LIN {X 0,Y 152.112,Z 664.807,A -85,B 0,C 180,E1 -25600.837,E2 -25600.837} C_VEL
LIN {X 0,Y 146.265,Z 675.889,A -85,B 0,C 180,E1 -25603.884,E2 -25603.884} C_VEL
LIN {X 0,Y 140.329,Z 686.128,A -85,B 0,C 180,E1 -25607.459,E2 -25607.459} C_VEL
LIN {X 0,Y 134.268,Z 696.183,A -85,B 0,C 180,E1 -25612.046,E2 -25612.046} C_VEL
LIN {X 0,Y 129.23,Z 704.605,A -85,B 0,C 180,E1 -25617.054,E2 -25617.054} C_VEL
LIN {X 0,Y 124.936,Z 712.522,A -85,B 0,C 180,E1 -25623.254,E2 -25623.254} C_VEL
LIN {X 0,Y 122.172,Z 718.854,A -85,B 0,C 180,E1 -25629.808,E2 -25629.808} C_VEL
LIN {X 0,Y 121.041,Z 723.776,A -85,B 0,C 180,E1 -25636.569,E2 -25636.569} C_VEL
LIN {X 0,Y 121.369,Z 727.342,A -85,B 0,C 180,E1 -25643.348,E2 -25643.348} C_VEL
LIN {X 0,Y 121.7,Z 728.339,A -85,B 0,C 180,E1 -25646.011,E2 -25646.011} C_VEL
LIN {X 0,Y 121.232,Z 728.844,A -85,B 0,C 180,E1 -25647.815,E2 -25647.815} C_VEL
LIN {X 0,Y 119.721,Z 729.035,A -85,B 0,C 180,E1 -25649.561,E2 -25649.561} C_VEL
LIN {X 0,Y 114.837,Z 728.936,A -85,B 0,C 180,E1 -25654.372,E2 -25654.372} C_VEL
LIN {X 0,Y 114.337,Z 728.882,A -85,B 0,C 180,E1 -25655.721,E2 -25655.721} C_VEL
LIN {X 0,Y 113.821,Z 728.676,A -85,B 0,C 180,E1 -25660.673,E2 -25660.673} C_VEL
LIN {X 0,Y 114.375,Z 727.382,A -85,B 0,C 180,E1 -25667.891,E2 -25667.891} C_VEL
LIN {X 0,Y 117.287,Z 724.46,A -85,B 0,C 180,E1 -25675.999,E2 -25675.999} C_VEL
LIN {X 0,Y 122.084,Z 720.301,A -85,B 0,C 180,E1 -25683.151,E2 -25683.151} C_VEL
LIN {X 0,Y 128.148,Z 715.223,A -85,B 0,C 180,E1 -25689.099,E2 -25689.099} C_VEL
LIN {X 0,Y 135.57,Z 708.791,A -85,B 0,C 180,E1 -25694.412,E2 -25694.412} C_VEL
LIN {X 0,Y 144.175,Z 700.89,A -85,B 0,C 180,E1 -25699.071,E2 -25699.071} C_VEL
LIN {X 0,Y 153.874,Z 691.31,A -85,B 0,C 180,E1 -25703.059,E2 -25703.059} C_VEL
LIN {X 0,Y 161.553,Z 682.701,A -85,B 0,C 180,E1 -25705.742,E2 -25705.742} C_VEL
LIN {X 0,Y 169.66,Z 672.712,A -85,B 0,C 180,E1 -25708.12,E2 -25708.12} C_VEL
LIN {X 0,Y 178.185,Z 660.946,A -85,B 0,C 180,E1 -25710.191,E2 -25710.191} C_VEL
LIN {X 0,Y 186.287,Z 648.041,A -85,B 0,C 180,E1 -25711.863,E2 -25711.863} C_VEL
LIN {X 0,Y 193.002,Z 635.336,A -85,B 0,C 180,E1 -25713.14,E2 -25713.14} C_VEL
LIN {X 0,Y 198.339,Z 623.513,A -85,B 0,C 180,E1 -25714.041,E2 -25714.041} C_VEL
LIN {X 0,Y 203.672,Z 608.798,A -85,B 0,C 180,E1 -25714.925,E2 -25714.925} C_VEL
LIN {X 0,Y 207.856,Z 593.51,A -85,B 0,C 180,E1 -25715.612,E2 -25715.612} C_VEL
LIN {X 0,Y 210.78,Z 577.845,A -85,B 0,C 180,E1 -25716.128,E2 -25716.128} C_VEL
LIN {X 0,Y 214.688,Z 540.152,A -85,B 0,C 180,E1 -25717.041,E2 -25717.041} C_VEL
LIN {X 0,Y 212.531,Z 531.894,A -85,B 0,C 180,E1 -25719.647,E2 -25719.647} C_VEL
LIN {X 0,Y 210.604,Z 524.936,A -85,B 0,C 180,E1 -25722.358,E2 -25722.358} C_VEL
LIN {X 0,Y 208.889,Z 519.075,A -85,B 0,C 180,E1 -25725.299,E2 -25725.299} C_VEL
LIN {X 0,Y 207.864,Z 515.191,A -85,B 0,C 180,E1 -25727.626,E2 -25727.626} C_VEL
LIN {X 0,Y 206.577,Z 509.756,A -85,B 0,C 180,E1 -25732.318,E2 -25732.318} C_VEL
LIN {X 0,Y 206.426,Z 508.775,A -85,B 0,C 180,E1 -25733.504,E2 -25733.504} C_VEL
LIN {X 0,Y 206.448,Z 508.658,A -85,B 0,C 180,E1 -25739.513,E2 -25739.513} C_VEL
LIN {X 0,Y 208.229,Z 512.983,A -85,B 0,C 180,E1 -25745.508,E2 -25745.508} C_VEL
LIN {X 0,Y 210.191,Z 517.111,A -85,B 0,C 180,E1 -25749.042,E2 -25749.042} C_VEL
LIN {X 0,Y 212.228,Z 521.339,A -85,B 0,C 180,E1 -25751.824,E2 -25751.824} C_VEL
LIN {X 0,Y 215.125,Z 527.412,A -85,B 0,C 180,E1 -25755.015,E2 -25755.015} C_VEL
LIN {X 0,Y 215.758,Z 528.889,A -85,B 0,C 180,E1 -25755.648,E2 -25755.648} C_VEL
LIN {X 0,Y 213.115,Z 556.855,A -85,B 0,C 180,E1 -25756.59,E2 -25756.59} C_VEL
LIN {X 0,Y 210.858,Z 570.576,A -85,B 0,C 180,E1 -25757.266,E2 -25757.266} C_VEL
LIN {X 0,Y 207.171,Z 585.652,A -85,B 0,C 180,E1 -25758.227,E2 -25758.227} C_VEL
LIN {X 0,Y 202.935,Z 598.669,A -85,B 0,C 180,E1 -25759.322,E2 -25759.322} C_VEL
LIN {X 0,Y 197.926,Z 611.211,A -85,B 0,C 180,E1 -25760.677,E2 -25760.677} C_VEL
LIN {X 0,Y 191.785,Z 623.736,A -85,B 0,C 180,E1 -25762.293,E2 -25762.293} C_VEL
LIN {X 0,Y 184.944,Z 635.502,A -85,B 0,C 180,E1 -25764.22,E2 -25764.22} C_VEL
LIN {X 0,Y 176.984,Z 647.191,A -85,B 0,C 180,E1 -25766.693,E2 -25766.693} C_VEL
LIN {X 0,Y 169.299,Z 656.934,A -85,B 0,C 180,E1 -25769.341,E2 -25769.341} C_VEL
LIN {X 0,Y 160.734,Z 666.373,A -85,B 0,C 180,E1 -25772.685,E2 -25772.685} C_VEL
LIN {X 0,Y 152.46,Z 674.345,A -85,B 0,C 180,E1 -25776.451,E2 -25776.451} C_VEL
LIN {X 0,Y 144.183,Z 681.32,A -85,B 0,C 180,E1 -25780.932,E2 -25780.932} C_VEL
LIN {X 0,Y 136.527,Z 686.987,A -85,B 0,C 180,E1 -25786.112,E2 -25786.112} C_VEL
LIN {X 0,Y 131.621,Z 690.179,A -85,B 0,C 180,E1 -25790.155,E2 -25790.155} C_VEL
LIN {X 0,Y 125.932,Z 693.387,A -85,B 0,C 180,E1 -25796.079,E2 -25796.079} C_VEL
LIN {X 0,Y 121.441,Z 695.394,A -85,B 0,C 180,E1 -25802.423,E2 -25802.423} C_VEL
LIN {X 0,Y 118.353,Z 696.242,A -85,B 0,C 180,E1 -25809.129,E2 -25809.129} C_VEL
LIN {X 0,Y 116.654,Z 695.972,A -85,B 0,C 180,E1 -25816.057,E2 -25816.057} C_VEL
LIN {X 0,Y 116.026,Z 694.601,A -85,B 0,C 180,E1 -25823.043,E2 -25823.043} C_VEL
LIN {X 0,Y 116.863,Z 692.077,A -85,B 0,C 180,E1 -25830.001,E2 -25830.001} C_VEL
LIN {X 0,Y 118.905,Z 688.408,A -85,B 0,C 180,E1 -25836.79,E2 -25836.79} C_VEL
LIN {X 0,Y 122.063,Z 683.523,A -85,B 0,C 180,E1 -25843.316,E2 -25843.316} C_VEL
LIN {X 0,Y 126.468,Z 677.262,A -85,B 0,C 180,E1 -25849.478,E2 -25849.478} C_VEL
LIN {X 0,Y 131.942,Z 669.449,A -85,B 0,C 180,E1 -25855.223,E2 -25855.223} C_VEL
LIN {X 0,Y 137.496,Z 661.145,A -85,B 0,C 180,E1 -25859.892,E2 -25859.892} C_VEL
LIN {X 0,Y 143.772,Z 651.153,A -85,B 0,C 180,E1 -25864.205,E2 -25864.205} C_VEL
LIN {X 0,Y 149.59,Z 640.955,A -85,B 0,C 180,E1 -25867.645,E2 -25867.645} C_VEL
LIN {X 0,Y 155.595,Z 628.801,A -85,B 0,C 180,E1 -25870.915,E2 -25870.915} C_VEL
LIN {X 0,Y 161.011,Z 616.564,A -85,B 0,C 180,E1 -25873.43,E2 -25873.43} C_VEL
LIN {X 0,Y 166.031,Z 603.169,A -85,B 0,C 180,E1 -25875.586,E2 -25875.586} C_VEL
LIN {X 0,Y 170.263,Z 589.275,A -85,B 0,C 180,E1 -25877.328,E2 -25877.328} C_VEL
LIN {X 0,Y 173.623,Z 575.007,A -85,B 0,C 180,E1 -25878.71,E2 -25878.71} C_VEL
LIN {X 0,Y 176.335,Z 559.317,A -85,B 0,C 180,E1 -25879.769,E2 -25879.769} C_VEL
LIN {X 0,Y 177.885,Z 543.275,A -85,B 0,C 180,E1 -25880.541,E2 -25880.541} C_VEL
LIN {X 0,Y 181.077,Z 501.444,A -85,B 0,C 180,E1 -25882,E2 -25882} C_VEL
LIN {X 0,Y 176.773,Z 492.406,A -85,B 0,C 180,E1 -25885.022,E2 -25885.022} C_VEL
LIN {X 0,Y 172.294,Z 483.86,A -85,B 0,C 180,E1 -25888.613,E2 -25888.613} C_VEL
LIN {X 0,Y 168.158,Z 476.667,A -85,B 0,C 180,E1 -25892.541,E2 -25892.541} C_VEL
LIN {X 0,Y 165.346,Z 472.291,A -85,B 0,C 180,E1 -25895.716,E2 -25895.716} C_VEL
LIN {X 0,Y 163.231,Z 468.887,A -85,B 0,C 180,E1 -25898.6,E2 -25898.6} C_VEL
LIN {X 0,Y 160.878,Z 465.055,A -85,B 0,C 180,E1 -25902.718,E2 -25902.718} C_VEL
LIN {X 0,Y 158.454,Z 461.541,A -85,B 0,C 180,E1 -25910.004,E2 -25910.004} C_VEL
LIN {X 0,Y 158.278,Z 459.994,A -85,B 0,C 180,E1 -25912.344,E2 -25912.344} C_VEL
LIN {X 0,Y 158.418,Z 459.872,A -85,B 0,C 180,E1 -25917.616,E2 -25917.616} C_VEL
LIN {X 0,Y 159.139,Z 462.833,A -85,B 0,C 180,E1 -25921.897,E2 -25921.897} C_VEL
LIN {X 0,Y 160.93,Z 464.889,A -85,B 0,C 180,E1 -25926.25,E2 -25926.25} C_VEL
LIN {X 0,Y 163.185,Z 468.728,A -85,B 0,C 180,E1 -25930.233,E2 -25930.233} C_VEL
LIN {X 0,Y 164.069,Z 470.08,A -85,B 0,C 180,E1 -25931.504,E2 -25931.504} C_VEL
LIN {X 0,Y 165.979,Z 474.343,A -85,B 0,C 180,E1 -25934.11,E2 -25934.11} C_VEL
LIN {X 0,Y 168.676,Z 480.782,A -85,B 0,C 180,E1 -25937.269,E2 -25937.269} C_VEL
LIN {X 0,Y 171.447,Z 487.752,A -85,B 0,C 180,E1 -25940.078,E2 -25940.078} C_VEL
LIN {X 0,Y 174.742,Z 497.166,A -85,B 0,C 180,E1 -25943.077,E2 -25943.077} C_VEL
LIN {X 0,Y 178.052,Z 507.617,A -85,B 0,C 180,E1 -25945.807,E2 -25945.807} C_VEL
LIN {X 0,Y 178.78,Z 510.414,A -85,B 0,C 180,E1 -25946.404,E2 -25946.404} C_VEL
LIN {X 0,Y 178.869,Z 533.313,A -85,B 0,C 180,E1 -25948.131,E2 -25948.131} C_VEL
LIN {X 0,Y 174.573,Z 581.759,A -85,B 0,C 180,E1 -25949.655,E2 -25949.655} C_VEL
LIN {X 0,Y 171.96,Z 597.666,A -85,B 0,C 180,E1 -25950.453,E2 -25950.453} C_VEL
LIN {X 0,Y 168.411,Z 612.372,A -85,B 0,C 180,E1 -25951.474,E2 -25951.474} C_VEL
LIN {X 0,Y 164.078,Z 626.316,A -85,B 0,C 180,E1 -25952.797,E2 -25952.797} C_VEL
LIN {X 0,Y 158.843,Z 639.968,A -85,B 0,C 180,E1 -25954.507,E2 -25954.507} C_VEL
LIN {X 0,Y 152.428,Z 653.818,A -85,B 0,C 180,E1 -25956.759,E2 -25956.759} C_VEL
LIN {X 0,Y 146.345,Z 665.337,A -85,B 0,C 180,E1 -25959.251,E2 -25959.251} C_VEL
LIN {X 0,Y 140.291,Z 676.167,A -85,B 0,C 180,E1 -25962.361,E2 -25962.361} C_VEL
LIN {X 0,Y 134.108,Z 686.187,A -85,B 0,C 180,E1 -25966.023,E2 -25966.023} C_VEL
LIN {X 0,Y 127.627,Z 696.341,A -85,B 0,C 180,E1 -25970.926,E2 -25970.926} C_VEL
LIN {X 0,Y 121.908,Z 705.397,A -85,B 0,C 180,E1 -25976.792,E2 -25976.792} C_VEL
LIN {X 0,Y 117.648,Z 712.863,A -85,B 0,C 180,E1 -25983.269,E2 -25983.269} C_VEL
LIN {X 0,Y 114.906,Z 718.974,A -85,B 0,C 180,E1 -25990.342,E2 -25990.342} C_VEL
LIN {X 0,Y 114.027,Z 722.601,A -85,B 0,C 180,E1 -25995.726,E2 -25995.726} C_VEL
LIN {X 0,Y 114.263,Z 726.206,A -85,B 0,C 180,E1 -26002.933,E2 -26002.933} C_VEL
LIN {X 0,Y 115.499,Z 728.454,A -85,B 0,C 180,E1 -26009.999,E2 -26009.999} C_VEL
LIN {X 0,Y 114.337,Z 728.882,A -85,B 0,C 180,E1 -26015.721,E2 -26015.721} C_VEL
LIN {X 0,Y 113.784,Z 728.846,A -85,B 0,C 180,E1 -26017.676,E2 -26017.676} C_VEL
LIN {X 0,Y 111.621,Z 728.326,A -85,B 0,C 180,E1 -26021.535,E2 -26021.535} C_VEL
LIN {X 0,Y 108.362,Z 726.846,A -85,B 0,C 180,E1 -26027.486,E2 -26027.486} C_VEL
LIN {X 0,Y 108.015,Z 725.981,A -85,B 0,C 180,E1 -26030.593,E2 -26030.593} C_VEL
LIN {X 0,Y 108.244,Z 725.674,A -85,B 0,C 180,E1 -26031.623,E2 -26031.623} C_VEL
LIN {X 0,Y 110.575,Z 723.732,A -85,B 0,C 180,E1 -26037.151,E2 -26037.151} C_VEL
LIN {X 0,Y 116.1,Z 719.409,A -85,B 0,C 180,E1 -26045.102,E2 -26045.102} C_VEL
LIN {X 0,Y 122.646,Z 714.362,A -85,B 0,C 180,E1 -26051.22,E2 -26051.22} C_VEL
LIN {X 0,Y 130.523,Z 707.987,A -85,B 0,C 180,E1 -26056.624,E2 -26056.624} C_VEL
LIN {X 0,Y 138.396,Z 701.205,A -85,B 0,C 180,E1 -26060.749,E2 -26060.749} C_VEL
LIN {X 0,Y 148.374,Z 691.91,A -85,B 0,C 180,E1 -26064.789,E2 -26064.789} C_VEL
LIN {X 0,Y 156.505,Z 683.356,A -85,B 0,C 180,E1 -26067.559,E2 -26067.559} C_VEL
LIN {X 0,Y 166.001,Z 672.212,A -85,B 0,C 180,E1 -26070.212,E2 -26070.212} C_VEL
LIN {X 0,Y 174.758,Z 660.554,A -85,B 0,C 180,E1 -26072.215,E2 -26072.215} C_VEL
LIN {X 0,Y 183.045,Z 647.785,A -85,B 0,C 180,E1 -26073.824,E2 -26073.824} C_VEL
LIN {X 0,Y 189.897,Z 635.255,A -85,B 0,C 180,E1 -26075.053,E2 -26075.053} C_VEL
LIN {X 0,Y 195.343,Z 623.545,A -85,B 0,C 180,E1 -26075.909,E2 -26075.909} C_VEL
LIN {X 0,Y 200.78,Z 609.126,A -85,B 0,C 180,E1 -26076.752,E2 -26076.752} C_VEL
LIN {X 0,Y 205.041,Z 594.319,A -85,B 0,C 180,E1 -26077.409,E2 -26077.409} C_VEL
LIN {X 0,Y 208.127,Z 579.032,A -85,B 0,C 180,E1 -26077.911,E2 -26077.911} C_VEL
LIN {X 0,Y 210.906,Z 554.927,A -85,B 0,C 180,E1 -26078.497,E2 -26078.497} C_VEL
LIN {X 0,Y 212.063,Z 543.415,A -85,B 0,C 180,E1 -26078.775,E2 -26078.775} C_VEL
LIN {X 0,Y 210.048,Z 535.02,A -85,B 0,C 180,E1 -26081.604,E2 -26081.604} C_VEL
LIN {X 0,Y 208.705,Z 529.937,A -85,B 0,C 180,E1 -26083.782,E2 -26083.782} C_VEL
LIN {X 0,Y 207.452,Z 525.087,A -85,B 0,C 180,E1 -26086.282,E2 -26086.282} C_VEL
LIN {X 0,Y 206.613,Z 521.553,A -85,B 0,C 180,E1 -26088.473,E2 -26088.473} C_VEL
LIN {X 0,Y 205.649,Z 516.707,A -85,B 0,C 180,E1 -26092.588,E2 -26092.588} C_VEL
LIN {X 0,Y 205.456,Z 515.784,A -85,B 0,C 180,E1 -26094.11,E2 -26094.11} C_VEL
LIN {X 0,Y 205.5,Z 515.62,A -85,B 0,C 180,E1 -26099.021,E2 -26099.021} C_VEL
LIN {X 0,Y 205.929,Z 517.273,A -85,B 0,C 180,E1 -26101.62,E2 -26101.62} C_VEL
LIN {X 0,Y 207.132,Z 519.832,A -85,B 0,C 180,E1 -26105.08,E2 -26105.08} C_VEL
LIN {X 0,Y 208.816,Z 523.632,A -85,B 0,C 180,E1 -26108.349,E2 -26108.349} C_VEL
LIN {X 0,Y 210.833,Z 528.018,A -85,B 0,C 180,E1 -26111.287,E2 -26111.287} C_VEL
LIN {X 0,Y 213.11,Z 533.062,A -85,B 0,C 180,E1 -26113.975,E2 -26113.975} C_VEL
LIN {X 0,Y 210.566,Z 558.418,A -85,B 0,C 180,E1 -26114.827,E2 -26114.827} C_VEL
LIN {X 0,Y 208.164,Z 572.425,A -85,B 0,C 180,E1 -26115.528,E2 -26115.528} C_VEL
LIN {X 0,Y 204.652,Z 586.243,A -85,B 0,C 180,E1 -26116.389,E2 -26116.389} C_VEL
LIN {X 0,Y 200.295,Z 599.365,A -85,B 0,C 180,E1 -26117.461,E2 -26117.461} C_VEL
LIN {X 0,Y 194.771,Z 612.768,A -85,B 0,C 180,E1 -26118.872,E2 -26118.872} C_VEL
LIN {X 0,Y 189.111,Z 623.995,A -85,B 0,C 180,E1 -26120.28,E2 -26120.28} C_VEL
LIN {X 0,Y 182.104,Z 635.823,A -85,B 0,C 180,E1 -26122.15,E2 -26122.15} C_VEL
LIN {X 0,Y 173.868,Z 647.633,A -85,B 0,C 180,E1 -26124.571,E2 -26124.571} C_VEL
LIN {X 0,Y 165.884,Z 657.476,A -85,B 0,C 180,E1 -26127.169,E2 -26127.169} C_VEL
LIN {X 0,Y 158.226,Z 665.783,A -85,B 0,C 180,E1 -26129.992,E2 -26129.992} C_VEL
LIN {X 0,Y 149.708,Z 673.835,A -85,B 0,C 180,E1 -26133.568,E2 -26133.568} C_VEL
LIN {X 0,Y 141.732,Z 680.433,A -85,B 0,C 180,E1 -26137.501,E2 -26137.501} C_VEL
LIN {X 0,Y 133.469,Z 686.463,A -85,B 0,C 180,E1 -26142.511,E2 -26142.511} C_VEL
LIN {X 0,Y 126.179,Z 691.039,A -85,B 0,C 180,E1 -26148.061,E2 -26148.061} C_VEL
LIN {X 0,Y 120.042,Z 694.301,A -85,B 0,C 180,E1 -26154.167,E2 -26154.167} C_VEL
LIN {X 0,Y 115.137,Z 696.359,A -85,B 0,C 180,E1 -26160.772,E2 -26160.772} C_VEL
LIN {X 0,Y 111.693,Z 697.26,A -85,B 0,C 180,E1 -26167.821,E2 -26167.821} C_VEL
LIN {X 0,Y 109.743,Z 697.031,A -85,B 0,C 180,E1 -26175.159,E2 -26175.159} C_VEL
LIN {X 0,Y 108.988,Z 695.69,A -85,B 0,C 180,E1 -26182.592,E2 -26182.592} C_VEL
LIN {X 0,Y 109.794,Z 693.218,A -85,B 0,C 180,E1 -26190.001,E2 -26190.001} C_VEL
LIN {X 0,Y 111.922,Z 689.6,A -85,B 0,C 180,E1 -26197.216,E2 -26197.216} C_VEL
LIN {X 0,Y 115.242,Z 684.772,A -85,B 0,C 180,E1 -26204.12,E2 -26204.12} C_VEL
LIN {X 0,Y 119.905,Z 678.569,A -85,B 0,C 180,E1 -26210.591,E2 -26210.591} C_VEL
LIN {X 0,Y 125.651,Z 670.828,A -85,B 0,C 180,E1 -26216.581,E2 -26216.581} C_VEL
LIN {X 0,Y 131.5,Z 662.597,A -85,B 0,C 180,E1 -26221.406,E2 -26221.406} C_VEL
LIN {X 0,Y 138.059,Z 652.696,A -85,B 0,C 180,E1 -26225.833,E2 -26225.833} C_VEL
LIN {X 0,Y 144.136,Z 642.602,A -85,B 0,C 180,E1 -26229.337,E2 -26229.337} C_VEL
LIN {X 0,Y 150.417,Z 630.569,A -85,B 0,C 180,E1 -26232.648,E2 -26232.648} C_VEL
LIN {X 0,Y 156.035,Z 618.496,A -85,B 0,C 180,E1 -26235.186,E2 -26235.186} C_VEL
LIN {X 0,Y 161.262,Z 605.302,A -85,B 0,C 180,E1 -26237.343,E2 -26237.343} C_VEL
LIN {X 0,Y 165.643,Z 591.684,A -85,B 0,C 180,E1 -26239.091,E2 -26239.091} C_VEL
LIN {X 0,Y 169.131,Z 577.782,A -85,B 0,C 180,E1 -26240.474,E2 -26240.474} C_VEL
LIN {X 0,Y 171.984,Z 562.633,A -85,B 0,C 180,E1 -26241.553,E2 -26241.553} C_VEL
LIN {X 0,Y 173.766,Z 547.313,A -85,B 0,C 180,E1 -26242.31,E2 -26242.31} C_VEL
LIN {X 0,Y 176.966,Z 507.169,A -85,B 0,C 180,E1 -26243.726,E2 -26243.726} C_VEL
LIN {X 0,Y 177.068,Z 504.448,A -85,B 0,C 180,E1 -26243.885,E2 -26243.885} C_VEL
LIN {X 0,Y 173.15,Z 496.062,A -85,B 0,C 180,E1 -26246.92,E2 -26246.92} C_VEL
LIN {X 0,Y 169.353,Z 488.56,A -85,B 0,C 180,E1 -26250.289,E2 -26250.289} C_VEL
LIN {X 0,Y 165.766,Z 482.228,A -85,B 0,C 180,E1 -26254.026,E2 -26254.026} C_VEL
LIN {X 0,Y 163.781,Z 478.872,A -85,B 0,C 180,E1 -26256.467,E2 -26256.467} C_VEL
LIN {X 0,Y 161.727,Z 475.429,A -85,B 0,C 180,E1 -26259.457,E2 -26259.457} C_VEL
LIN {X 0,Y 159.517,Z 471.62,A -85,B 0,C 180,E1 -26263.687,E2 -26263.687} C_VEL
LIN {X 0,Y 157.609,Z 468.874,A -85,B 0,C 180,E1 -26269.725,E2 -26269.725} C_VEL
LIN {X 0,Y 157.362,Z 467.006,A -85,B 0,C 180,E1 -26272.945,E2 -26272.945} C_VEL
LIN {X 0,Y 157.502,Z 467.081,A -85,B 0,C 180,E1 -26277.442,E2 -26277.442} C_VEL
LIN {X 0,Y 158.254,Z 469.982,A -85,B 0,C 180,E1 -26281.908,E2 -26281.908} C_VEL
LIN {X 0,Y 159.761,Z 471.82,A -85,B 0,C 180,E1 -26285.728,E2 -26285.728} C_VEL
LIN {X 0,Y 161.89,Z 475.532,A -85,B 0,C 180,E1 -26289.684,E2 -26289.684} C_VEL
LIN {X 0,Y 163.035,Z 477.817,A -85,B 0,C 180,E1 -26291.46,E2 -26291.46} C_VEL
LIN {X 0,Y 164.162,Z 480.658,A -85,B 0,C 180,E1 -26293.106,E2 -26293.106} C_VEL
LIN {X 0,Y 166.379,Z 486.256,A -85,B 0,C 180,E1 -26295.936,E2 -26295.936} C_VEL
LIN {X 0,Y 169.023,Z 493.456,A -85,B 0,C 180,E1 -26298.877,E2 -26298.877} C_VEL
LIN {X 0,Y 171.838,Z 502.041,A -85,B 0,C 180,E1 -26301.676,E2 -26301.676} C_VEL
LIN {X 0,Y 175.081,Z 513.049,A -85,B 0,C 180,E1 -26304.595,E2 -26304.595} C_VEL
LIN {X 0,Y 174.908,Z 535.394,A -85,B 0,C 180,E1 -26306.266,E2 -26306.266} C_VEL
LIN {X 0,Y 170.777,Z 580.315,A -85,B 0,C 180,E1 -26307.655,E2 -26307.655} C_VEL
LIN {X 0,Y 168.047,Z 596.417,A -85,B 0,C 180,E1 -26308.43,E2 -26308.43} C_VEL
LIN {X 0,Y 164.413,Z 611.138,A -85,B 0,C 180,E1 -26309.431,E2 -26309.431} C_VEL
LIN {X 0,Y 160.298,Z 624.113,A -85,B 0,C 180,E1 -26310.636,E2 -26310.636} C_VEL
LIN {X 0,Y 154.899,Z 638.009,A -85,B 0,C 180,E1 -26312.324,E2 -26312.324} C_VEL
LIN {X 0,Y 148.631,Z 651.257,A -85,B 0,C 180,E1 -26314.4,E2 -26314.4} C_VEL
LIN {X 0,Y 141.884,Z 663.665,A -85,B 0,C 180,E1 -26316.992,E2 -26316.992} C_VEL
LIN {X 0,Y 135.513,Z 674.596,A -85,B 0,C 180,E1 -26320.096,E2 -26320.096} C_VEL
LIN {X 0,Y 129.022,Z 684.714,A -85,B 0,C 180,E1 -26323.801,E2 -26323.801} C_VEL
LIN {X 0,Y 123.209,Z 693.309,A -85,B 0,C 180,E1 -26327.862,E2 -26327.862} C_VEL
LIN {X 0,Y 117.382,Z 701.932,A -85,B 0,C 180,E1 -26333.22,E2 -26333.22} C_VEL
LIN {X 0,Y 112.19,Z 709.964,A -85,B 0,C 180,E1 -26339.923,E2 -26339.923} C_VEL
LIN {X 0,Y 108.725,Z 716.409,A -85,B 0,C 180,E1 -26347.179,E2 -26347.179} C_VEL
LIN {X 0,Y 107.026,Z 721.409,A -85,B 0,C 180,E1 -26354.771,E2 -26354.771} C_VEL
LIN {X 0,Y 107.142,Z 725.065,A -85,B 0,C 180,E1 -26362.46,E2 -26362.46} C_VEL
LIN {X 0,Y 108.393,Z 727.372,A -85,B 0,C 180,E1 -26369.999,E2 -26369.999} C_VEL
LIN {X 0,Y 107.083,Z 727.865,A -85,B 0,C 180,E1 -26377.541,E2 -26377.541} C_VEL
LIN {X 0,Y 106.902,Z 727.158,A -85,B 0,C 180,E1 -26385.244,E2 -26385.244} C_VEL
LIN {X 0,Y 108.244,Z 725.674,A -85,B 0,C 180,E1 -26391.623,E2 -26391.623} C_VEL
LIN {X 0,Y 108.72,Z 724.686,A -85,B 0,C 180,E1 -26394.691,E2 -26394.691} C_VEL
LIN {X 0,Y 108.395,Z 722.594,A -85,B 0,C 180,E1 -26399.809,E2 -26399.809} C_VEL
LIN {X 0,Y 108.624,Z 720.558,A -85,B 0,C 180,E1 -26403.868,E2 -26403.868} C_VEL
LIN {X 0,Y 109.916,Z 718.836,A -85,B 0,C 180,E1 -26406.758,E2 -26406.758} C_VEL
LIN {X 0,Y 110.658,Z 718.231,A -85,B 0,C 180,E1 -26407.654,E2 -26407.654} C_VEL
LIN {X 0,Y 117.317,Z 713.505,A -85,B 0,C 180,E1 -26413.542,E2 -26413.542} C_VEL
LIN {X 0,Y 125.684,Z 707.187,A -85,B 0,C 180,E1 -26419.012,E2 -26419.012} C_VEL
LIN {X 0,Y 135.238,Z 699.421,A -85,B 0,C 180,E1 -26423.654,E2 -26423.654} C_VEL
LIN {X 0,Y 144.38,Z 691.245,A -85,B 0,C 180,E1 -26427.102,E2 -26427.102} C_VEL
LIN {X 0,Y 152.598,Z 682.98,A -85,B 0,C 180,E1 -26429.762,E2 -26429.762} C_VEL
LIN {X 0,Y 161.119,Z 673.488,A -85,B 0,C 180,E1 -26432.038,E2 -26432.038} C_VEL
LIN {X 0,Y 170.797,Z 661.236,A -85,B 0,C 180,E1 -26434.168,E2 -26434.168} C_VEL
LIN {X 0,Y 179.248,Z 648.81,A -85,B 0,C 180,E1 -26435.721,E2 -26435.721} C_VEL
LIN {X 0,Y 187.016,Z 635.164,A -85,B 0,C 180,E1 -26437.023,E2 -26437.023} C_VEL
LIN {X 0,Y 192.564,Z 623.575,A -85,B 0,C 180,E1 -26437.831,E2 -26437.831} C_VEL
LIN {X 0,Y 198.093,Z 609.452,A -85,B 0,C 180,E1 -26438.633,E2 -26438.633} C_VEL
LIN {X 0,Y 202.628,Z 594.364,A -85,B 0,C 180,E1 -26439.285,E2 -26439.285} C_VEL
LIN {X 0,Y 205.909,Z 578.826,A -85,B 0,C 180,E1 -26439.784,E2 -26439.784} C_VEL
LIN {X 0,Y 208.479,Z 557.906,A -85,B 0,C 180,E1 -26440.285,E2 -26440.285} C_VEL
LIN {X 0,Y 209.647,Z 546.785,A -85,B 0,C 180,E1 -26440.528,E2 -26440.528} C_VEL
LIN {X 0,Y 207.883,Z 538.858,A -85,B 0,C 180,E1 -26443.419,E2 -26443.419} C_VEL
LIN {X 0,Y 206.241,Z 531.798,A -85,B 0,C 180,E1 -26446.866,E2 -26446.866} C_VEL
LIN {X 0,Y 205.418,Z 527.904,A -85,B 0,C 180,E1 -26449.31,E2 -26449.31} C_VEL
LIN {X 0,Y 204.675,Z 523.442,A -85,B 0,C 180,E1 -26453.208,E2 -26453.208} C_VEL
LIN {X 0,Y 204.589,Z 522.852,A -85,B 0,C 180,E1 -26454.085,E2 -26454.085} C_VEL
LIN {X 0,Y 204.66,Z 522.742,A -85,B 0,C 180,E1 -26459.263,E2 -26459.263} C_VEL
LIN {X 0,Y 206.043,Z 526.707,A -85,B 0,C 180,E1 -26464.647,E2 -26464.647} C_VEL
LIN {X 0,Y 207.551,Z 530.322,A -85,B 0,C 180,E1 -26467.785,E2 -26467.785} C_VEL
LIN {X 0,Y 209.656,Z 535.161,A -85,B 0,C 180,E1 -26471.014,E2 -26471.014} C_VEL
LIN {X 0,Y 210.607,Z 537.691,A -85,B 0,C 180,E1 -26472.276,E2 -26472.276} C_VEL
LIN {X 0,Y 208.197,Z 560.164,A -85,B 0,C 180,E1 -26473.034,E2 -26473.034} C_VEL
LIN {X 0,Y 205.63,Z 574.297,A -85,B 0,C 180,E1 -26473.741,E2 -26473.741} C_VEL
LIN {X 0,Y 201.971,Z 588.128,A -85,B 0,C 180,E1 -26474.59,E2 -26474.59} C_VEL
LIN {X 0,Y 197.133,Z 602.066,A -85,B 0,C 180,E1 -26475.732,E2 -26475.732} C_VEL
LIN {X 0,Y 191.228,Z 615.598,A -85,B 0,C 180,E1 -26477.155,E2 -26477.155} C_VEL
LIN {X 0,Y 184.595,Z 627.95,A -85,B 0,C 180,E1 -26478.735,E2 -26478.735} C_VEL
LIN {X 0,Y 177.471,Z 639.17,A -85,B 0,C 180,E1 -26480.561,E2 -26480.561} C_VEL
LIN {X 0,Y 169.605,Z 649.838,A -85,B 0,C 180,E1 -26482.788,E2 -26482.788} C_VEL
LIN {X 0,Y 161.414,Z 659.44,A -85,B 0,C 180,E1 -26485.349,E2 -26485.349} C_VEL
LIN {X 0,Y 152.15,Z 668.832,A -85,B 0,C 180,E1 -26488.646,E2 -26488.646} C_VEL
LIN {X 0,Y 144.623,Z 675.552,A -85,B 0,C 180,E1 -26491.747,E2 -26491.747} C_VEL
LIN {X 0,Y 135.2,Z 682.857,A -85,B 0,C 180,E1 -26496.324,E2 -26496.324} C_VEL
LIN {X 0,Y 128.708,Z 687.265,A -85,B 0,C 180,E1 -26500.145,E2 -26500.145} C_VEL
LIN {X 0,Y 120.932,Z 691.899,A -85,B 0,C 180,E1 -26505.786,E2 -26505.786} C_VEL
LIN {X 0,Y 114.292,Z 695.217,A -85,B 0,C 180,E1 -26512.057,E2 -26512.057} C_VEL
LIN {X 0,Y 108.939,Z 697.326,A -85,B 0,C 180,E1 -26518.931,E2 -26518.931} C_VEL
LIN {X 0,Y 105.117,Z 698.277,A -85,B 0,C 180,E1 -26526.352,E2 -26526.352} C_VEL
LIN {X 0,Y 102.864,Z 698.076,A -85,B 0,C 180,E1 -26534.142,E2 -26534.142} C_VEL
LIN {X 0,Y 101.96,Z 696.779,A -85,B 0,C 180,E1 -26542.078,E2 -26542.078} C_VEL
LIN {X 0,Y 102.729,Z 694.356,A -85,B 0,C 180,E1 -26550.002,E2 -26550.002} C_VEL
LIN {X 0,Y 104.947,Z 690.789,A -85,B 0,C 180,E1 -26557.698,E2 -26557.698} C_VEL
LIN {X 0,Y 108.446,Z 686.017,A -85,B 0,C 180,E1 -26565.025,E2 -26565.025} C_VEL
LIN {X 0,Y 113.367,Z 679.875,A -85,B 0,C 180,E1 -26571.837,E2 -26571.837} C_VEL
LIN {X 0,Y 119.437,Z 672.199,A -85,B 0,C 180,E1 -26578.083,E2 -26578.083} C_VEL
LIN {X 0,Y 125.6,Z 664.041,A -85,B 0,C 180,E1 -26583.064,E2 -26583.064} C_VEL
LIN {X 0,Y 132.472,Z 654.228,A -85,B 0,C 180,E1 -26587.598,E2 -26587.598} C_VEL
LIN {X 0,Y 138.834,Z 644.223,A -85,B 0,C 180,E1 -26591.154,E2 -26591.154} C_VEL
LIN {X 0,Y 145.4,Z 632.32,A -85,B 0,C 180,E1 -26594.497,E2 -26594.497} C_VEL
LIN {X 0,Y 151.212,Z 620.368,A -85,B 0,C 180,E1 -26597.056,E2 -26597.056} C_VEL
LIN {X 0,Y 156.626,Z 607.354,A -85,B 0,C 180,E1 -26599.218,E2 -26599.218} C_VEL
LIN {X 0,Y 161.484,Z 593.017,A -85,B 0,C 180,E1 -26601.073,E2 -26601.073} C_VEL
LIN {X 0,Y 165.426,Z 577.946,A -85,B 0,C 180,E1 -26602.553,E2 -26602.553} C_VEL
LIN {X 0,Y 168.409,Z 562.39,A -85,B 0,C 180,E1 -26603.617,E2 -26603.617} C_VEL
LIN {X 0,Y 170.178,Z 546.885,A -85,B 0,C 180,E1 -26604.362,E2 -26604.362} C_VEL
LIN {X 0,Y 173.343,Z 507.8,A -85,B 0,C 180,E1 -26605.774,E2 -26605.774} C_VEL
LIN {X 0,Y 169.281,Z 498.823,A -85,B 0,C 180,E1 -26609.305,E2 -26609.305} C_VEL
LIN {X 0,Y 166.035,Z 492.321,A -85,B 0,C 180,E1 -26612.58,E2 -26612.58} C_VEL
LIN {X 0,Y 162.659,Z 486.034,A -85,B 0,C 180,E1 -26616.682,E2 -26616.682} C_VEL
LIN {X 0,Y 160.349,Z 482.108,A -85,B 0,C 180,E1 -26620.181,E2 -26620.181} C_VEL
LIN {X 0,Y 158.377,Z 478.512,A -85,B 0,C 180,E1 -26624.228,E2 -26624.228} C_VEL
LIN {X 0,Y 156.635,Z 475.708,A -85,B 0,C 180,E1 -26630.34,E2 -26630.34} C_VEL
LIN {X 0,Y 156.466,Z 474.001,A -85,B 0,C 180,E1 -26633.552,E2 -26633.552} C_VEL
LIN {X 0,Y 156.593,Z 474.269,A -85,B 0,C 180,E1 -26637.276,E2 -26637.276} C_VEL
LIN {X 0,Y 157.37,Z 477.122,A -85,B 0,C 180,E1 -26641.919,E2 -26641.919} C_VEL
LIN {X 0,Y 158.563,Z 478.622,A -85,B 0,C 180,E1 -26645.085,E2 -26645.085} C_VEL
LIN {X 0,Y 160.972,Z 483.055,A -85,B 0,C 180,E1 -26649.74,E2 -26649.74} C_VEL
LIN {X 0,Y 162.272,Z 486.508,A -85,B 0,C 180,E1 -26651.871,E2 -26651.871} C_VEL
LIN {X 0,Y 164.307,Z 492.109,A -85,B 0,C 180,E1 -26654.741,E2 -26654.741} C_VEL
LIN {X 0,Y 166.726,Z 499.277,A -85,B 0,C 180,E1 -26657.695,E2 -26657.695} C_VEL
LIN {X 0,Y 169.426,Z 508.237,A -85,B 0,C 180,E1 -26660.625,E2 -26660.625} C_VEL
LIN {X 0,Y 171.556,Z 516.284,A -85,B 0,C 180,E1 -26662.764,E2 -26662.764} C_VEL
LIN {X 0,Y 171.229,Z 536.211,A -85,B 0,C 180,E1 -26664.268,E2 -26664.268} C_VEL
LIN {X 0,Y 167.019,Z 579.936,A -85,B 0,C 180,E1 -26665.607,E2 -26665.607} C_VEL
LIN {X 0,Y 164.23,Z 595.762,A -85,B 0,C 180,E1 -26666.365,E2 -26666.365} C_VEL
LIN {X 0,Y 160.294,Z 611.04,A -85,B 0,C 180,E1 -26667.397,E2 -26667.397} C_VEL
LIN {X 0,Y 156.059,Z 623.907,A -85,B 0,C 180,E1 -26668.578,E2 -26668.578} C_VEL
LIN {X 0,Y 150.498,Z 637.643,A -85,B 0,C 180,E1 -26670.241,E2 -26670.241} C_VEL
LIN {X 0,Y 143.622,Z 651.56,A -85,B 0,C 180,E1 -26672.424,E2 -26672.424} C_VEL
LIN {X 0,Y 136.417,Z 664.191,A -85,B 0,C 180,E1 -26675.13,E2 -26675.13} C_VEL
LIN {X 0,Y 128.658,Z 676.669,A -85,B 0,C 180,E1 -26678.884,E2 -26678.884} C_VEL
LIN {X 0,Y 121.983,Z 686.312,A -85,B 0,C 180,E1 -26682.728,E2 -26682.728} C_VEL
LIN {X 0,Y 115.108,Z 695.83,A -85,B 0,C 180,E1 -26687.808,E2 -26687.808} C_VEL
LIN {X 0,Y 109.303,Z 703.772,A -85,B 0,C 180,E1 -26693.504,E2 -26693.504} C_VEL
LIN {X 0,Y 104.729,Z 710.571,A -85,B 0,C 180,E1 -26700.003,E2 -26700.003} C_VEL
LIN {X 0,Y 101.401,Z 716.524,A -85,B 0,C 180,E1 -26707.591,E2 -26707.591} C_VEL
LIN {X 0,Y 99.893,Z 721.246,A -85,B 0,C 180,E1 -26715.743,E2 -26715.743} C_VEL
LIN {X 0,Y 100.025,Z 723.922,A -85,B 0,C 180,E1 -26721.92,E2 -26721.92} C_VEL
LIN {X 0,Y 101.285,Z 726.288,A -85,B 0,C 180,E1 -26729.998,E2 -26729.998} C_VEL
LIN {X 0,Y 100.521,Z 726.711,A -85,B 0,C 180,E1 -26734.008,E2 -26734.008} C_VEL
LIN {X 0,Y 99.722,Z 726.622,A -85,B 0,C 180,E1 -26742.204,E2 -26742.204} C_VEL
LIN {X 0,Y 100.742,Z 725.394,A -85,B 0,C 180,E1 -26750.412,E2 -26750.412} C_VEL
LIN {X 0,Y 103.933,Z 722.95,A -85,B 0,C 180,E1 -26758.472,E2 -26758.472} C_VEL
LIN {X 0,Y 110.282,Z 718.509,A -85,B 0,C 180,E1 -26767.255,E2 -26767.255} C_VEL
LIN {X 0,Y 110.658,Z 718.231,A -85,B 0,C 180,E1 -26767.654,E2 -26767.654} C_VEL
LIN {X 0,Y 112.664,Z 716.386,A -85,B 0,C 180,E1 -26770.338,E2 -26770.338} C_VEL
LIN {X 0,Y 114.893,Z 712.97,A -85,B 0,C 180,E1 -26774.898,E2 -26774.898} C_VEL
LIN {X 0,Y 117.767,Z 709.211,A -85,B 0,C 180,E1 -26779.185,E2 -26779.185} C_VEL
LIN {X 0,Y 120.666,Z 706.701,A -85,B 0,C 180,E1 -26781.348,E2 -26781.348} C_VEL
LIN {X 0,Y 129.801,Z 699.734,A -85,B 0,C 180,E1 -26785.655,E2 -26785.655} C_VEL
LIN {X 0,Y 139.227,Z 691.844,A -85,B 0,C 180,E1 -26789.103,E2 -26789.103} C_VEL
LIN {X 0,Y 148.934,Z 682.6,A -85,B 0,C 180,E1 -26792.076,E2 -26792.076} C_VEL
LIN {X 0,Y 157.899,Z 672.941,A -85,B 0,C 180,E1 -26794.326,E2 -26794.326} C_VEL
LIN {X 0,Y 167.827,Z 660.803,A -85,B 0,C 180,E1 -26796.349,E2 -26796.349} C_VEL
LIN {X 0,Y 176.444,Z 648.487,A -85,B 0,C 180,E1 -26797.826,E2 -26797.826} C_VEL
LIN {X 0,Y 184.361,Z 635.004,A -85,B 0,C 180,E1 -26799.055,E2 -26799.055} C_VEL
LIN {X 0,Y 190.811,Z 621.834,A -85,B 0,C 180,E1 -26799.915,E2 -26799.915} C_VEL
LIN {X 0,Y 196.426,Z 607.523,A -85,B 0,C 180,E1 -26800.673,E2 -26800.673} C_VEL
LIN {X 0,Y 200.966,Z 592.392,A -85,B 0,C 180,E1 -26801.278,E2 -26801.278} C_VEL
LIN {X 0,Y 204.17,Z 577.144,A -85,B 0,C 180,E1 -26801.738,E2 -26801.738} C_VEL
LIN {X 0,Y 206.928,Z 554.742,A -85,B 0,C 180,E1 -26802.234,E2 -26802.234} C_VEL
LIN {X 0,Y 207.384,Z 550.17,A -85,B 0,C 180,E1 -26802.37,E2 -26802.37} C_VEL
LIN {X 0,Y 206.007,Z 543.205,A -85,B 0,C 180,E1 -26805.089,E2 -26805.089} C_VEL
LIN {X 0,Y 204.853,Z 537.548,A -85,B 0,C 180,E1 -26808.032,E2 -26808.032} C_VEL
LIN {X 0,Y 204.325,Z 534.604,A -85,B 0,C 180,E1 -26809.91,E2 -26809.91} C_VEL
LIN {X 0,Y 203.728,Z 530.188,A -85,B 0,C 180,E1 -26813.812,E2 -26813.812} C_VEL
LIN {X 0,Y 203.697,Z 529.672,A -85,B 0,C 180,E1 -26818.567,E2 -26818.567} C_VEL
LIN {X 0,Y 204.877,Z 533.236,A -85,B 0,C 180,E1 -26823.935,E2 -26823.935} C_VEL
LIN {X 0,Y 206.328,Z 537.069,A -85,B 0,C 180,E1 -26827.255,E2 -26827.255} C_VEL
LIN {X 0,Y 208.176,Z 541.617,A -85,B 0,C 180,E1 -26830.306,E2 -26830.306} C_VEL
LIN {X 0,Y 208.329,Z 542.017,A -85,B 0,C 180,E1 -26830.531,E2 -26830.531} C_VEL
LIN {X 0,Y 206.012,Z 562.102,A -85,B 0,C 180,E1 -26831.215,E2 -26831.215} C_VEL
LIN {X 0,Y 203.287,Z 576.239,A -85,B 0,C 180,E1 -26831.924,E2 -26831.924} C_VEL
LIN {X 0,Y 199.883,Z 588.74,A -85,B 0,C 180,E1 -26832.666,E2 -26832.666} C_VEL
LIN {X 0,Y 195.29,Z 601.76,A -85,B 0,C 180,E1 -26833.682,E2 -26833.682} C_VEL
LIN {X 0,Y 189.128,Z 615.755,A -85,B 0,C 180,E1 -26835.078,E2 -26835.078} C_VEL
LIN {X 0,Y 183.165,Z 626.825,A -85,B 0,C 180,E1 -26836.423,E2 -26836.423} C_VEL
LIN {X 0,Y 175.552,Z 638.804,A -85,B 0,C 180,E1 -26838.239,E2 -26838.239} C_VEL
LIN {X 0,Y 166.942,Z 650.28,A -85,B 0,C 180,E1 -26840.504,E2 -26840.504} C_VEL
LIN {X 0,Y 158.288,Z 660.167,A -85,B 0,C 180,E1 -26843.052,E2 -26843.052} C_VEL
LIN {X 0,Y 148.837,Z 669.458,A -85,B 0,C 180,E1 -26846.217,E2 -26846.217} C_VEL
LIN {X 0,Y 140.983,Z 676.243,A -85,B 0,C 180,E1 -26849.269,E2 -26849.269} C_VEL
LIN {X 0,Y 131.061,Z 683.627,A -85,B 0,C 180,E1 -26853.785,E2 -26853.785} C_VEL
LIN {X 0,Y 121.817,Z 689.523,A -85,B 0,C 180,E1 -26859.11,E2 -26859.11} C_VEL
LIN {X 0,Y 115.884,Z 692.759,A -85,B 0,C 180,E1 -26863.305,E2 -26863.305} C_VEL
LIN {X 0,Y 108.719,Z 696.132,A -85,B 0,C 180,E1 -26869.73,E2 -26869.73} C_VEL
LIN {X 0,Y 102.869,Z 698.293,A -85,B 0,C 180,E1 -26876.871,E2 -26876.871} C_VEL
LIN {X 0,Y 98.597,Z 699.294,A -85,B 0,C 180,E1 -26884.682,E2 -26884.682} C_VEL
LIN {X 0,Y 96.027,Z 699.117,A -85,B 0,C 180,E1 -26892.979,E2 -26892.979} C_VEL
LIN {X 0,Y 94.941,Z 697.867,A -85,B 0,C 180,E1 -26901.488,E2 -26901.488} C_VEL
LIN {X 0,Y 95.648,Z 695.496,A -85,B 0,C 180,E1 -26910.002,E2 -26910.002} C_VEL
LIN {X 0,Y 97.981,Z 691.977,A -85,B 0,C 180,E1 -26918.249,E2 -26918.249} C_VEL
LIN {X 0,Y 101.682,Z 687.261,A -85,B 0,C 180,E1 -26926.051,E2 -26926.051} C_VEL
LIN {X 0,Y 106.906,Z 681.177,A -85,B 0,C 180,E1 -26933.232,E2 -26933.232} C_VEL
LIN {X 0,Y 113.325,Z 673.567,A -85,B 0,C 180,E1 -26939.745,E2 -26939.745} C_VEL
LIN {X 0,Y 119.809,Z 665.486,A -85,B 0,C 180,E1 -26944.886,E2 -26944.886} C_VEL
LIN {X 0,Y 127.017,Z 655.76,A -85,B 0,C 180,E1 -26949.517,E2 -26949.517} C_VEL
LIN {X 0,Y 133.664,Z 645.812,A -85,B 0,C 180,E1 -26953.121,E2 -26953.121} C_VEL
LIN {X 0,Y 140.541,Z 634.026,A -85,B 0,C 180,E1 -26956.477,E2 -26956.477} C_VEL
LIN {X 0,Y 146.553,Z 622.214,A -85,B 0,C 180,E1 -26959.051,E2 -26959.051} C_VEL
LIN {X 0,Y 152.167,Z 609.391,A -85,B 0,C 180,E1 -26961.205,E2 -26961.205} C_VEL
LIN {X 0,Y 157.217,Z 595.313,A -85,B 0,C 180,E1 -26963.04,E2 -26963.04} C_VEL
LIN {X 0,Y 161.306,Z 580.645,A -85,B 0,C 180,E1 -26964.508,E2 -26964.508} C_VEL
LIN {X 0,Y 164.402,Z 565.768,A -85,B 0,C 180,E1 -26965.564,E2 -26965.564} C_VEL
LIN {X 0,Y 166.43,Z 550.44,A -85,B 0,C 180,E1 -26966.331,E2 -26966.331} C_VEL
LIN {X 0,Y 169.758,Z 511.024,A -85,B 0,C 180,E1 -26967.793,E2 -26967.793} C_VEL
LIN {X 0,Y 166.026,Z 502.521,A -85,B 0,C 180,E1 -26971.437,E2 -26971.437} C_VEL
LIN {X 0,Y 162.689,Z 495.659,A -85,B 0,C 180,E1 -26975.318,E2 -26975.318} C_VEL
LIN {X 0,Y 160.252,Z 491.169,A -85,B 0,C 180,E1 -26978.756,E2 -26978.756} C_VEL
LIN {X 0,Y 158.855,Z 488.578,A -85,B 0,C 180,E1 -26981.172,E2 -26981.172} C_VEL
LIN {X 0,Y 157.194,Z 485.351,A -85,B 0,C 180,E1 -26984.917,E2 -26984.917} C_VEL
LIN {X 0,Y 155.658,Z 482.391,A -85,B 0,C 180,E1 -26991.215,E2 -26991.215} C_VEL
LIN {X 0,Y 155.594,Z 481.067,A -85,B 0,C 180,E1 -26993.567,E2 -26993.567} C_VEL
LIN {X 0,Y 155.678,Z 481.221,A -85,B 0,C 180,E1 -26996.804,E2 -26996.804} C_VEL
LIN {X 0,Y 156.35,Z 484.028,A -85,B 0,C 180,E1 -27001.448,E2 -27001.448} C_VEL
LIN {X 0,Y 157.405,Z 485.456,A -85,B 0,C 180,E1 -27004.481,E2 -27004.481} C_VEL
LIN {X 0,Y 159.52,Z 489.653,A -85,B 0,C 180,E1 -27008.91,E2 -27008.91} C_VEL
LIN {X 0,Y 160.563,Z 492.757,A -85,B 0,C 180,E1 -27010.8,E2 -27010.8} C_VEL
LIN {X 0,Y 162.608,Z 498.841,A -85,B 0,C 180,E1 -27013.94,E2 -27013.94} C_VEL
LIN {X 0,Y 164.999,Z 506.855,A -85,B 0,C 180,E1 -27017.107,E2 -27017.107} C_VEL
LIN {X 0,Y 167.591,Z 516.621,A -85,B 0,C 180,E1 -27020.14,E2 -27020.14} C_VEL
LIN {X 0,Y 168.178,Z 519.006,A -85,B 0,C 180,E1 -27020.785,E2 -27020.785} C_VEL
LIN {X 0,Y 167.869,Z 535.702,A -85,B 0,C 180,E1 -27022.135,E2 -27022.135} C_VEL
LIN {X 0,Y 163.576,Z 578.906,A -85,B 0,C 180,E1 -27023.438,E2 -27023.438} C_VEL
LIN {X 0,Y 160.784,Z 594.401,A -85,B 0,C 180,E1 -27024.153,E2 -27024.153} C_VEL
LIN {X 0,Y 156.748,Z 609.775,A -85,B 0,C 180,E1 -27025.16,E2 -27025.16} C_VEL
LIN {X 0,Y 152.031,Z 623.655,A -85,B 0,C 180,E1 -27026.408,E2 -27026.408} C_VEL
LIN {X 0,Y 146.307,Z 637.26,A -85,B 0,C 180,E1 -27028.036,E2 -27028.036} C_VEL
LIN {X 0,Y 139.216,Z 651.044,A -85,B 0,C 180,E1 -27030.173,E2 -27030.173} C_VEL
LIN {X 0,Y 131.749,Z 663.586,A -85,B 0,C 180,E1 -27032.843,E2 -27032.843} C_VEL
LIN {X 0,Y 124.257,Z 675.128,A -85,B 0,C 180,E1 -27036.294,E2 -27036.294} C_VEL
LIN {X 0,Y 116.098,Z 686.323,A -85,B 0,C 180,E1 -27040.827,E2 -27040.827} C_VEL
LIN {X 0,Y 108.889,Z 695.683,A -85,B 0,C 180,E1 -27046.065,E2 -27046.065} C_VEL
LIN {X 0,Y 102.768,Z 703.489,A -85,B 0,C 180,E1 -27052.012,E2 -27052.012} C_VEL
LIN {X 0,Y 97.268,Z 711.183,A -85,B 0,C 180,E1 -27060.116,E2 -27060.116} C_VEL
LIN {X 0,Y 94.07,Z 716.633,A -85,B 0,C 180,E1 -27068.064,E2 -27068.064} C_VEL
LIN {X 0,Y 92.788,Z 721.059,A -85,B 0,C 180,E1 -27076.865,E2 -27076.865} C_VEL
LIN {X 0,Y 93.391,Z 724.158,A -85,B 0,C 180,E1 -27085.683,E2 -27085.683} C_VEL
LIN {X 0,Y 94.174,Z 725.204,A -85,B 0,C 180,E1 -27089.998,E2 -27089.998} C_VEL
LIN {X 0,Y 93.406,Z 725.646,A -85,B 0,C 180,E1 -27094.313,E2 -27094.313} C_VEL
LIN {X 0,Y 92.71,Z 725.595,A -85,B 0,C 180,E1 -27103.143,E2 -27103.143} C_VEL
LIN {X 0,Y 94.021,Z 724.387,A -85,B 0,C 180,E1 -27111.945,E2 -27111.945} C_VEL
LIN {X 0,Y 97.55,Z 722.063,A -85,B 0,C 180,E1 -27120.283,E2 -27120.283} C_VEL
LIN {X 0,Y 104.29,Z 717.805,A -85,B 0,C 180,E1 -27129.301,E2 -27129.301} C_VEL
LIN {X 0,Y 111.97,Z 712.802,A -85,B 0,C 180,E1 -27135.909,E2 -27135.909} C_VEL
LIN {X 0,Y 120.666,Z 706.701,A -85,B 0,C 180,E1 -27141.348,E2 -27141.348} C_VEL
LIN {X 0,Y 123.716,Z 704.084,A -85,B 0,C 180,E1 -27143.383,E2 -27143.383} C_VEL
LIN {X 0,Y 131.548,Z 695.014,A -85,B 0,C 180,E1 -27149.917,E2 -27149.917} C_VEL
LIN {X 0,Y 134.327,Z 692.347,A -85,B 0,C 180,E1 -27151.235,E2 -27151.235} C_VEL
LIN {X 0,Y 135.616,Z 691.249,A -85,B 0,C 180,E1 -27151.663,E2 -27151.663} C_VEL
LIN {X 0,Y 144.382,Z 683.242,A -85,B 0,C 180,E1 -27154.22,E2 -27154.22} C_VEL
LIN {X 0,Y 153.415,Z 674.055,A -85,B 0,C 180,E1 -27156.372,E2 -27156.372} C_VEL
LIN {X 0,Y 162.729,Z 663.318,A -85,B 0,C 180,E1 -27158.204,E2 -27158.204} C_VEL
LIN {X 0,Y 171.465,Z 651.708,A -85,B 0,C 180,E1 -27159.646,E2 -27159.646} C_VEL
LIN {X 0,Y 179.551,Z 639.136,A -85,B 0,C 180,E1 -27160.78,E2 -27160.78} C_VEL
LIN {X 0,Y 185.184,Z 628.657,A -85,B 0,C 180,E1 -27161.576,E2 -27161.576} C_VEL
LIN {X 0,Y 190.924,Z 616.256,A -85,B 0,C 180,E1 -27162.257,E2 -27162.257} C_VEL
LIN {X 0,Y 196.228,Z 601.91,A -85,B 0,C 180,E1 -27162.898,E2 -27162.898} C_VEL
LIN {X 0,Y 200.505,Z 586.491,A -85,B 0,C 180,E1 -27163.401,E2 -27163.401} C_VEL
LIN {X 0,Y 203.329,Z 571.239,A -85,B 0,C 180,E1 -27163.812,E2 -27163.812} C_VEL
LIN {X 0,Y 205.351,Z 553.791,A -85,B 0,C 180,E1 -27164.198,E2 -27164.198} C_VEL
LIN {X 0,Y 204.425,Z 548.53,A -85,B 0,C 180,E1 -27166.424,E2 -27166.424} C_VEL
LIN {X 0,Y 203.624,Z 543.769,A -85,B 0,C 180,E1 -27168.932,E2 -27168.932} C_VEL
LIN {X 0,Y 203.208,Z 541.018,A -85,B 0,C 180,E1 -27170.739,E2 -27170.739} C_VEL
LIN {X 0,Y 202.813,Z 537.015,A -85,B 0,C 180,E1 -27174.283,E2 -27174.283} C_VEL
LIN {X 0,Y 202.843,Z 536.798,A -85,B 0,C 180,E1 -27178.76,E2 -27178.76} C_VEL
LIN {X 0,Y 203.868,Z 540.274,A -85,B 0,C 180,E1 -27183.645,E2 -27183.645} C_VEL
LIN {X 0,Y 205.164,Z 543.909,A -85,B 0,C 180,E1 -27186.801,E2 -27186.801} C_VEL
LIN {X 0,Y 206.198,Z 546.675,A -85,B 0,C 180,E1 -27188.717,E2 -27188.717} C_VEL
LIN {X 0,Y 203.939,Z 564.718,A -85,B 0,C 180,E1 -27189.381,E2 -27189.381} C_VEL
LIN {X 0,Y 200.735,Z 579.852,A -85,B 0,C 180,E1 -27190.142,E2 -27190.142} C_VEL
LIN {X 0,Y 196.369,Z 594.263,A -85,B 0,C 180,E1 -27191.038,E2 -27191.038} C_VEL
LIN {X 0,Y 191.371,Z 607.142,A -85,B 0,C 180,E1 -27192.11,E2 -27192.11} C_VEL
LIN {X 0,Y 185.524,Z 619.382,A -85,B 0,C 180,E1 -27193.34,E2 -27193.34} C_VEL
LIN {X 0,Y 178.939,Z 630.867,A -85,B 0,C 180,E1 -27194.732,E2 -27194.732} C_VEL
LIN {X 0,Y 170.964,Z 642.583,A -85,B 0,C 180,E1 -27196.556,E2 -27196.556} C_VEL
LIN {X 0,Y 161.606,Z 654.238,A -85,B 0,C 180,E1 -27198.945,E2 -27198.945} C_VEL
LIN {X 0,Y 152.043,Z 664.342,A -85,B 0,C 180,E1 -27201.703,E2 -27201.703} C_VEL
LIN {X 0,Y 141.649,Z 673.656,A -85,B 0,C 180,E1 -27205.117,E2 -27205.117} C_VEL
LIN {X 0,Y 132.392,Z 680.811,A -85,B 0,C 180,E1 -27208.756,E2 -27208.756} C_VEL
LIN {X 0,Y 122.314,Z 687.492,A -85,B 0,C 180,E1 -27213.581,E2 -27213.581} C_VEL
LIN {X 0,Y 113.206,Z 692.591,A -85,B 0,C 180,E1 -27219.106,E2 -27219.106} C_VEL
LIN {X 0,Y 107.062,Z 695.49,A -85,B 0,C 180,E1 -27223.776,E2 -27223.776} C_VEL
LIN {X 0,Y 99.985,Z 698.297,A -85,B 0,C 180,E1 -27230.76,E2 -27230.76} C_VEL
LIN {X 0,Y 94.345,Z 699.929,A -85,B 0,C 180,E1 -27238.574,E2 -27238.574} C_VEL
LIN {X 0,Y 90.475,Z 700.366,A -85,B 0,C 180,E1 -27247.148,E2 -27247.148} C_VEL
LIN {X 0,Y 88.423,Z 699.682,A -85,B 0,C 180,E1 -27256.207,E2 -27256.207} C_VEL
LIN {X 0,Y 88.042,Z 697.932,A -85,B 0,C 180,E1 -27265.423,E2 -27265.423} C_VEL
LIN {X 0,Y 89.622,Z 695.041,A -85,B 0,C 180,E1 -27274.499,E2 -27274.499} C_VEL
LIN {X 0,Y 92.85,Z 690.982,A -85,B 0,C 180,E1 -27283.126,E2 -27283.126} C_VEL
LIN {X 0,Y 97.548,Z 685.671,A -85,B 0,C 180,E1 -27291.116,E2 -27291.116} C_VEL
LIN {X 0,Y 103.77,Z 678.912,A -85,B 0,C 180,E1 -27298.301,E2 -27298.301} C_VEL
LIN {X 0,Y 111.125,Z 670.517,A -85,B 0,C 180,E1 -27304.695,E2 -27304.695} C_VEL
LIN {X 0,Y 118.431,Z 661.605,A -85,B 0,C 180,E1 -27309.638,E2 -27309.638} C_VEL
LIN {X 0,Y 126.326,Z 650.867,A -85,B 0,C 180,E1 -27314.061,E2 -27314.061} C_VEL
LIN {X 0,Y 133.437,Z 639.871,A -85,B 0,C 180,E1 -27317.508,E2 -27317.508} C_VEL
LIN {X 0,Y 140.166,Z 627.836,A -85,B 0,C 180,E1 -27320.436,E2 -27320.436} C_VEL
LIN {X 0,Y 146.617,Z 614.501,A -85,B 0,C 180,E1 -27322.836,E2 -27322.836} C_VEL
LIN {X 0,Y 151.842,Z 601.452,A -85,B 0,C 180,E1 -27324.663,E2 -27324.663} C_VEL
LIN {X 0,Y 156.433,Z 587.077,A -85,B 0,C 180,E1 -27326.216,E2 -27326.216} C_VEL
LIN {X 0,Y 160.065,Z 572.015,A -85,B 0,C 180,E1 -27327.419,E2 -27327.419} C_VEL
LIN {X 0,Y 162.671,Z 556.199,A -85,B 0,C 180,E1 -27328.28,E2 -27328.28} C_VEL
LIN {X 0,Y 166.073,Z 518.695,A -85,B 0,C 180,E1 -27329.683,E2 -27329.683} C_VEL
LIN {X 0,Y 166.443,Z 514.661,A -85,B 0,C 180,E1 -27329.816,E2 -27329.816} C_VEL
LIN {X 0,Y 163.216,Z 506.881,A -85,B 0,C 180,E1 -27333.378,E2 -27333.378} C_VEL
LIN {X 0,Y 160.18,Z 500.534,A -85,B 0,C 180,E1 -27337.37,E2 -27337.37} C_VEL
LIN {X 0,Y 157.892,Z 495.777,A -85,B 0,C 180,E1 -27341.251,E2 -27341.251} C_VEL
LIN {X 0,Y 156.157,Z 492.298,A -85,B 0,C 180,E1 -27345.295,E2 -27345.295} C_VEL
LIN {X 0,Y 154.749,Z 489.424,A -85,B 0,C 180,E1 -27351.498,E2 -27351.498} C_VEL
LIN {X 0,Y 154.712,Z 488.079,A -85,B 0,C 180,E1 -27354.132,E2 -27354.132} C_VEL
LIN {X 0,Y 154.775,Z 488.36,A -85,B 0,C 180,E1 -27356.593,E2 -27356.593} C_VEL
LIN {X 0,Y 155.47,Z 491.139,A -85,B 0,C 180,E1 -27361.456,E2 -27361.456} C_VEL
LIN {X 0,Y 156.278,Z 492.328,A -85,B 0,C 180,E1 -27363.908,E2 -27363.908} C_VEL
LIN {X 0,Y 158.079,Z 496.208,A -85,B 0,C 180,E1 -27368.026,E2 -27368.026} C_VEL
LIN {X 0,Y 159.033,Z 499.432,A -85,B 0,C 180,E1 -27369.94,E2 -27369.94} C_VEL
LIN {X 0,Y 160.671,Z 504.73,A -85,B 0,C 180,E1 -27372.713,E2 -27372.713} C_VEL
LIN {X 0,Y 162.71,Z 512.365,A -85,B 0,C 180,E1 -27375.741,E2 -27375.741} C_VEL
LIN {X 0,Y 164.982,Z 521.955,A -85,B 0,C 180,E1 -27378.732,E2 -27378.732} C_VEL
LIN {X 0,Y 164.639,Z 536.512,A -85,B 0,C 180,E1 -27379.968,E2 -27379.968} C_VEL
LIN {X 0,Y 160.383,Z 577.957,A -85,B 0,C 180,E1 -27381.195,E2 -27381.195} C_VEL
LIN {X 0,Y 157.591,Z 593.04,A -85,B 0,C 180,E1 -27381.851,E2 -27381.851} C_VEL
LIN {X 0,Y 153.47,Z 608.526,A -85,B 0,C 180,E1 -27382.839,E2 -27382.839} C_VEL
LIN {X 0,Y 148.973,Z 621.44,A -85,B 0,C 180,E1 -27383.931,E2 -27383.931} C_VEL
LIN {X 0,Y 143.817,Z 633.668,A -85,B 0,C 180,E1 -27385.305,E2 -27385.305} C_VEL
LIN {X 0,Y 137.228,Z 646.641,A -85,B 0,C 180,E1 -27387.147,E2 -27387.147} C_VEL
LIN {X 0,Y 129.363,Z 659.73,A -85,B 0,C 180,E1 -27389.63,E2 -27389.63} C_VEL
LIN {X 0,Y 122.667,Z 669.863,A -85,B 0,C 180,E1 -27392.32,E2 -27392.32} C_VEL
LIN {X 0,Y 115.132,Z 680.274,A -85,B 0,C 180,E1 -27396.019,E2 -27396.019} C_VEL
LIN {X 0,Y 107.352,Z 689.997,A -85,B 0,C 180,E1 -27400.672,E2 -27400.672} C_VEL
LIN {X 0,Y 99.87,Z 698.962,A -85,B 0,C 180,E1 -27406.676,E2 -27406.676} C_VEL
LIN {X 0,Y 93.989,Z 706.045,A -85,B 0,C 180,E1 -27413.258,E2 -27413.258} C_VEL
LIN {X 0,Y 89.099,Z 712.659,A -85,B 0,C 180,E1 -27421.752,E2 -27421.752} C_VEL
LIN {X 0,Y 86.322,Z 717.815,A -85,B 0,C 180,E1 -27430.993,E2 -27430.993} C_VEL
LIN {X 0,Y 85.811,Z 721.634,A -85,B 0,C 180,E1 -27440.571,E2 -27440.571} C_VEL
LIN {X 0,Y 87.057,Z 724.118,A -85,B 0,C 180,E1 -27449.998,E2 -27449.998} C_VEL
LIN {X 0,Y 86.29,Z 724.58,A -85,B 0,C 180,E1 -27454.67,E2 -27454.67} C_VEL
LIN {X 0,Y 85.711,Z 724.566,A -85,B 0,C 180,E1 -27464.238,E2 -27464.238} C_VEL
LIN {X 0,Y 87.38,Z 723.383,A -85,B 0,C 180,E1 -27473.71,E2 -27473.71} C_VEL
LIN {X 0,Y 91.394,Z 721.105,A -85,B 0,C 180,E1 -27482.564,E2 -27482.564} C_VEL
LIN {X 0,Y 97.395,Z 717.709,A -85,B 0,C 180,E1 -27490.496,E2 -27490.496} C_VEL
LIN {X 0,Y 105.159,Z 713.147,A -85,B 0,C 180,E1 -27497.316,E2 -27497.316} C_VEL
LIN {X 0,Y 114.305,Z 707.308,A -85,B 0,C 180,E1 -27503.059,E2 -27503.059} C_VEL
LIN {X 0,Y 124.537,Z 700.044,A -85,B 0,C 180,E1 -27507.828,E2 -27507.828} C_VEL
LIN {X 0,Y 135.616,Z 691.249,A -85,B 0,C 180,E1 -27511.663,E2 -27511.663} C_VEL
LIN {X 0,Y 139.19,Z 687.897,A -85,B 0,C 180,E1 -27513.035,E2 -27513.035} C_VEL
LIN {X 0,Y 143.869,Z 682.146,A -85,B 0,C 180,E1 -27515.706,E2 -27515.706} C_VEL
LIN {X 0,Y 148.587,Z 676.025,A -85,B 0,C 180,E1 -27518.133,E2 -27518.133} C_VEL
LIN {X 0,Y 152.097,Z 672.039,A -85,B 0,C 180,E1 -27519.123,E2 -27519.123} C_VEL
LIN {X 0,Y 161.842,Z 660.896,A -85,B 0,C 180,E1 -27520.813,E2 -27520.813} C_VEL
LIN {X 0,Y 170.774,Z 649.015,A -85,B 0,C 180,E1 -27522.109,E2 -27522.109} C_VEL
LIN {X 0,Y 178.951,Z 636.089,A -85,B 0,C 180,E1 -27523.185,E2 -27523.185} C_VEL
LIN {X 0,Y 185.586,Z 623.672,A -85,B 0,C 180,E1 -27523.924,E2 -27523.924} C_VEL
LIN {X 0,Y 191.793,Z 609.32,A -85,B 0,C 180,E1 -27524.611,E2 -27524.611} C_VEL
LIN {X 0,Y 196.848,Z 594.147,A -85,B 0,C 180,E1 -27525.182,E2 -27525.182} C_VEL
LIN {X 0,Y 200.469,Z 579.215,A -85,B 0,C 180,E1 -27525.588,E2 -27525.588} C_VEL
LIN {X 0,Y 202.945,Z 562.82,A -85,B 0,C 180,E1 -27525.949,E2 -27525.949} C_VEL
LIN {X 0,Y 203.526,Z 557.537,A -85,B 0,C 180,E1 -27526.071,E2 -27526.071} C_VEL
LIN {X 0,Y 202.72,Z 551.967,A -85,B 0,C 180,E1 -27528.692,E2 -27528.692} C_VEL
LIN {X 0,Y 202.188,Z 547.819,A -85,B 0,C 180,E1 -27531.257,E2 -27531.257} C_VEL
LIN {X 0,Y 201.916,Z 544.052,A -85,B 0,C 180,E1 -27534.508,E2 -27534.508} C_VEL
LIN {X 0,Y 201.947,Z 543.766,A -85,B 0,C 180,E1 -27538.505,E2 -27538.505} C_VEL
LIN {X 0,Y 202.865,Z 547.309,A -85,B 0,C 180,E1 -27543.352,E2 -27543.352} C_VEL
LIN {X 0,Y 204.053,Z 550.859,A -85,B 0,C 180,E1 -27546.427,E2 -27546.427} C_VEL
LIN {X 0,Y 204.308,Z 551.556,A -85,B 0,C 180,E1 -27546.957,E2 -27546.957} C_VEL
LIN {X 0,Y 202.026,Z 567.674,A -85,B 0,C 180,E1 -27547.527,E2 -27547.527} C_VEL
LIN {X 0,Y 198.655,Z 582.433,A -85,B 0,C 180,E1 -27548.263,E2 -27548.263} C_VEL
LIN {X 0,Y 194.173,Z 596.478,A -85,B 0,C 180,E1 -27549.126,E2 -27549.126} C_VEL
LIN {X 0,Y 189.189,Z 608.806,A -85,B 0,C 180,E1 -27550.139,E2 -27550.139} C_VEL
LIN {X 0,Y 182.671,Z 621.856,A -85,B 0,C 180,E1 -27551.403,E2 -27551.403} C_VEL
LIN {X 0,Y 175.672,Z 633.495,A -85,B 0,C 180,E1 -27552.809,E2 -27552.809} C_VEL
LIN {X 0,Y 167.087,Z 645.488,A -85,B 0,C 180,E1 -27554.674,E2 -27554.674} C_VEL
LIN {X 0,Y 157.895,Z 656.347,A -85,B 0,C 180,E1 -27556.876,E2 -27556.876} C_VEL
LIN {X 0,Y 147.759,Z 666.519,A -85,B 0,C 180,E1 -27559.629,E2 -27559.629} C_VEL
LIN {X 0,Y 137.327,Z 675.41,A -85,B 0,C 180,E1 -27562.906,E2 -27562.906} C_VEL
LIN {X 0,Y 128.679,Z 681.808,A -85,B 0,C 180,E1 -27566.126,E2 -27566.126} C_VEL
LIN {X 0,Y 118.479,Z 688.267,A -85,B 0,C 180,E1 -27570.675,E2 -27570.675} C_VEL
LIN {X 0,Y 108.808,Z 693.422,A -85,B 0,C 180,E1 -27576.163,E2 -27576.163} C_VEL
LIN {X 0,Y 102.216,Z 696.379,A -85,B 0,C 180,E1 -27580.863,E2 -27580.863} C_VEL
LIN {X 0,Y 94.551,Z 699.237,A -85,B 0,C 180,E1 -27588.016,E2 -27588.016} C_VEL
LIN {X 0,Y 88.326,Z 700.906,A -85,B 0,C 180,E1 -27596.156,E2 -27596.156} C_VEL
LIN {X 0,Y 83.926,Z 701.384,A -85,B 0,C 180,E1 -27605.25,E2 -27605.25} C_VEL
LIN {X 0,Y 81.524,Z 700.748,A -85,B 0,C 180,E1 -27615.014,E2 -27615.014} C_VEL
LIN {X 0,Y 80.996,Z 699.044,A -85,B 0,C 180,E1 -27625.024,E2 -27625.024} C_VEL
LIN {X 0,Y 82.57,Z 696.207,A -85,B 0,C 180,E1 -27634.884,E2 -27634.884} C_VEL
LIN {X 0,Y 86.022,Z 692.198,A -85,B 0,C 180,E1 -27644.189,E2 -27644.189} C_VEL
LIN {X 0,Y 91.039,Z 686.936,A -85,B 0,C 180,E1 -27652.706,E2 -27652.706} C_VEL
LIN {X 0,Y 97.677,Z 680.231,A -85,B 0,C 180,E1 -27660.243,E2 -27660.243} C_VEL
LIN {X 0,Y 105.458,Z 671.922,A -85,B 0,C 180,E1 -27666.855,E2 -27666.855} C_VEL
LIN {X 0,Y 113.143,Z 663.078,A -85,B 0,C 180,E1 -27671.894,E2 -27671.894} C_VEL
LIN {X 0,Y 121.414,Z 652.449,A -85,B 0,C 180,E1 -27676.349,E2 -27676.349} C_VEL
LIN {X 0,Y 128.847,Z 641.548,A -85,B 0,C 180,E1 -27679.786,E2 -27679.786} C_VEL
LIN {X 0,Y 135.829,Z 629.642,A -85,B 0,C 180,E1 -27682.705,E2 -27682.705} C_VEL
LIN {X 0,Y 142.538,Z 616.489,A -85,B 0,C 180,E1 -27685.056,E2 -27685.056} C_VEL
LIN {X 0,Y 148.624,Z 601.83,A -85,B 0,C 180,E1 -27687.071,E2 -27687.071} C_VEL
LIN {X 0,Y 153.372,Z 587.274,A -85,B 0,C 180,E1 -27688.589,E2 -27688.589} C_VEL
LIN {X 0,Y 156.899,Z 573.018,A -85,B 0,C 180,E1 -27689.7,E2 -27689.7} C_VEL
LIN {X 0,Y 159.561,Z 557.604,A -85,B 0,C 180,E1 -27690.514,E2 -27690.514} C_VEL
LIN {X 0,Y 163.027,Z 521.065,A -85,B 0,C 180,E1 -27691.875,E2 -27691.875} C_VEL
LIN {X 0,Y 163.212,Z 517.955,A -85,B 0,C 180,E1 -27692.072,E2 -27692.072} C_VEL
LIN {X 0,Y 160.697,Z 511.715,A -85,B 0,C 180,E1 -27695.213,E2 -27695.213} C_VEL
LIN {X 0,Y 158.314,Z 506.327,A -85,B 0,C 180,E1 -27698.75,E2 -27698.75} C_VEL
LIN {X 0,Y 156.262,Z 501.932,A -85,B 0,C 180,E1 -27702.664,E2 -27702.664} C_VEL
LIN {X 0,Y 154.964,Z 499.053,A -85,B 0,C 180,E1 -27706.144,E2 -27706.144} C_VEL
LIN {X 0,Y 153.82,Z 496.125,A -85,B 0,C 180,E1 -27712.369,E2 -27712.369} C_VEL
LIN {X 0,Y 153.839,Z 495.163,A -85,B 0,C 180,E1 -27714.099,E2 -27714.099} C_VEL
LIN {X 0,Y 153.878,Z 495.483,A -85,B 0,C 180,E1 -27716.399,E2 -27716.399} C_VEL
LIN {X 0,Y 154.6,Z 498.295,A -85,B 0,C 180,E1 -27721.514,E2 -27721.514} C_VEL
LIN {X 0,Y 155.207,Z 499.292,A -85,B 0,C 180,E1 -27723.447,E2 -27723.447} C_VEL
LIN {X 0,Y 156.744,Z 502.936,A -85,B 0,C 180,E1 -27727.272,E2 -27727.272} C_VEL
LIN {X 0,Y 158.432,Z 509.279,A -85,B 0,C 180,E1 -27730.785,E2 -27730.785} C_VEL
LIN {X 0,Y 160.13,Z 516.218,A -85,B 0,C 180,E1 -27733.725,E2 -27733.725} C_VEL
LIN {X 0,Y 162.018,Z 524.874,A -85,B 0,C 180,E1 -27736.607,E2 -27736.607} C_VEL
LIN {X 0,Y 161.974,Z 528.841,A -85,B 0,C 180,E1 -27737.028,E2 -27737.028} C_VEL
LIN {X 0,Y 161.578,Z 538.332,A -85,B 0,C 180,E1 -27737.766,E2 -27737.766} C_VEL
LIN {X 0,Y 157.408,Z 577.09,A -85,B 0,C 180,E1 -27738.849,E2 -27738.849} C_VEL
LIN {X 0,Y 154.476,Z 592.464,A -85,B 0,C 180,E1 -27739.505,E2 -27739.505} C_VEL
LIN {X 0,Y 150.443,Z 607.266,A -85,B 0,C 180,E1 -27740.41,E2 -27740.41} C_VEL
LIN {X 0,Y 145.442,Z 621.212,A -85,B 0,C 180,E1 -27741.536,E2 -27741.536} C_VEL
LIN {X 0,Y 140.136,Z 633.279,A -85,B 0,C 180,E1 -27742.85,E2 -27742.85} C_VEL
LIN {X 0,Y 133.368,Z 646.145,A -85,B 0,C 180,E1 -27744.632,E2 -27744.632} C_VEL
LIN {X 0,Y 125.253,Z 659.144,A -85,B 0,C 180,E1 -27747.033,E2 -27747.033} C_VEL
LIN {X 0,Y 117.602,Z 670.12,A -85,B 0,C 180,E1 -27749.942,E2 -27749.942} C_VEL
LIN {X 0,Y 109.764,Z 680.323,A -85,B 0,C 180,E1 -27753.657,E2 -27753.657} C_VEL
LIN {X 0,Y 101.153,Z 690.399,A -85,B 0,C 180,E1 -27758.704,E2 -27758.704} C_VEL
LIN {X 0,Y 93.737,Z 698.677,A -85,B 0,C 180,E1 -27764.579,E2 -27764.579} C_VEL
LIN {X 0,Y 88.298,Z 704.729,A -85,B 0,C 180,E1 -27770.449,E2 -27770.449} C_VEL
LIN {X 0,Y 82.797,Z 711.401,A -85,B 0,C 180,E1 -27779.382,E2 -27779.382} C_VEL
LIN {X 0,Y 79.496,Z 716.607,A -85,B 0,C 180,E1 -27789.289,E2 -27789.289} C_VEL
LIN {X 0,Y 78.708,Z 720.485,A -85,B 0,C 180,E1 -27799.711,E2 -27799.711} C_VEL
LIN {X 0,Y 79.932,Z 723.03,A -85,B 0,C 180,E1 -27809.998,E2 -27809.998} C_VEL
LIN {X 0,Y 79.179,Z 723.515,A -85,B 0,C 180,E1 -27815.09,E2 -27815.09} C_VEL
LIN {X 0,Y 78.767,Z 723.532,A -85,B 0,C 180,E1 -27825.524,E2 -27825.524} C_VEL
LIN {X 0,Y 80.833,Z 722.378,A -85,B 0,C 180,E1 -27835.765,E2 -27835.765} C_VEL
LIN {X 0,Y 85.402,Z 720.148,A -85,B 0,C 180,E1 -27845.17,E2 -27845.17} C_VEL
LIN {X 0,Y 92.02,Z 716.799,A -85,B 0,C 180,E1 -27853.419,E2 -27853.419} C_VEL
LIN {X 0,Y 100.422,Z 712.293,A -85,B 0,C 180,E1 -27860.335,E2 -27860.335} C_VEL
LIN {X 0,Y 110.127,Z 706.5,A -85,B 0,C 180,E1 -27866.055,E2 -27866.055} C_VEL
LIN {X 0,Y 120.885,Z 699.291,A -85,B 0,C 180,E1 -27870.694,E2 -27870.694} C_VEL
LIN {X 0,Y 131.582,Z 691.19,A -85,B 0,C 180,E1 -27874.166,E2 -27874.166} C_VEL
LIN {X 0,Y 141.43,Z 682.614,A -85,B 0,C 180,E1 -27876.819,E2 -27876.819} C_VEL
LIN {X 0,Y 152.097,Z 672.039,A -85,B 0,C 180,E1 -27879.123,E2 -27879.123} C_VEL
LIN {X 0,Y 155.618,Z 667.965,A -85,B 0,C 180,E1 -27880.044,E2 -27880.044} C_VEL
LIN {X 0,Y 160.434,Z 661.147,A -85,B 0,C 180,E1 -27882.011,E2 -27882.011} C_VEL
LIN {X 0,Y 165.104,Z 653.964,A -85,B 0,C 180,E1 -27883.76,E2 -27883.76} C_VEL
LIN {X 0,Y 168.288,Z 649.327,A -85,B 0,C 180,E1 -27884.358,E2 -27884.358} C_VEL
LIN {X 0,Y 176.209,Z 637.383,A -85,B 0,C 180,E1 -27885.275,E2 -27885.275} C_VEL
LIN {X 0,Y 182.907,Z 625.36,A -85,B 0,C 180,E1 -27885.968,E2 -27885.968} C_VEL
LIN {X 0,Y 188.774,Z 612.663,A -85,B 0,C 180,E1 -27886.553,E2 -27886.553} C_VEL
LIN {X 0,Y 194.225,Z 597.873,A -85,B 0,C 180,E1 -27887.082,E2 -27887.082} C_VEL
LIN {X 0,Y 198.425,Z 582.478,A -85,B 0,C 180,E1 -27887.494,E2 -27887.494} C_VEL
LIN {X 0,Y 201.272,Z 566.473,A -85,B 0,C 180,E1 -27887.867,E2 -27887.867} C_VEL
LIN {X 0,Y 201.903,Z 561.327,A -85,B 0,C 180,E1 -27888.009,E2 -27888.009} C_VEL
LIN {X 0,Y 201.27,Z 555.599,A -85,B 0,C 180,E1 -27891.122,E2 -27891.122} C_VEL
LIN {X 0,Y 201.012,Z 551.219,A -85,B 0,C 180,E1 -27894.672,E2 -27894.672} C_VEL
LIN {X 0,Y 201.049,Z 550.788,A -85,B 0,C 180,E1 -27898.248,E2 -27898.248} C_VEL
LIN {X 0,Y 201.821,Z 554.108,A -85,B 0,C 180,E1 -27902.87,E2 -27902.87} C_VEL
LIN {X 0,Y 202.532,Z 556.607,A -85,B 0,C 180,E1 -27905.133,E2 -27905.133} C_VEL
LIN {X 0,Y 200.045,Z 571.775,A -85,B 0,C 180,E1 -27905.705,E2 -27905.705} C_VEL
LIN {X 0,Y 196.55,Z 585.758,A -85,B 0,C 180,E1 -27906.383,E2 -27906.383} C_VEL
LIN {X 0,Y 191.31,Z 600.943,A -85,B 0,C 180,E1 -27907.326,E2 -27907.326} C_VEL
LIN {X 0,Y 185.607,Z 613.962,A -85,B 0,C 180,E1 -27908.435,E2 -27908.435} C_VEL
LIN {X 0,Y 178.254,Z 627.386,A -85,B 0,C 180,E1 -27909.725,E2 -27909.725} C_VEL
LIN {X 0,Y 170.197,Z 639.588,A -85,B 0,C 180,E1 -27911.283,E2 -27911.283} C_VEL
LIN {X 0,Y 161.726,Z 650.4,A -85,B 0,C 180,E1 -27913.056,E2 -27913.056} C_VEL
LIN {X 0,Y 151.303,Z 661.656,A -85,B 0,C 180,E1 -27915.466,E2 -27915.466} C_VEL
LIN {X 0,Y 140.646,Z 671.344,A -85,B 0,C 180,E1 -27918.309,E2 -27918.309} C_VEL
LIN {X 0,Y 130.328,Z 679.33,A -85,B 0,C 180,E1 -27921.539,E2 -27921.539} C_VEL
LIN {X 0,Y 120.4,Z 685.862,A -85,B 0,C 180,E1 -27925.214,E2 -27925.214} C_VEL
LIN {X 0,Y 109.745,Z 691.825,A -85,B 0,C 180,E1 -27930.177,E2 -27930.177} C_VEL
LIN {X 0,Y 102.293,Z 695.341,A -85,B 0,C 180,E1 -27934.471,E2 -27934.471} C_VEL
LIN {X 0,Y 93.334,Z 698.877,A -85,B 0,C 180,E1 -27941.154,E2 -27941.154} C_VEL
LIN {X 0,Y 85.676,Z 701.183,A -85,B 0,C 180,E1 -27948.99,E2 -27948.99} C_VEL
LIN {X 0,Y 79.716,Z 702.281,A -85,B 0,C 180,E1 -27958.067,E2 -27958.067} C_VEL
LIN {X 0,Y 75.814,Z 702.243,A -85,B 0,C 180,E1 -27968.238,E2 -27968.238} C_VEL
LIN {X 0,Y 73.964,Z 701.132,A -85,B 0,C 180,E1 -27979.047,E2 -27979.047} C_VEL
LIN {X 0,Y 74.435,Z 698.912,A -85,B 0,C 180,E1 -27990.002,E2 -27990.002} C_VEL
LIN {X 0,Y 77.157,Z 695.54,A -85,B 0,C 180,E1 -28000.498,E2 -28000.498} C_VEL
LIN {X 0,Y 81.646,Z 690.972,A -85,B 0,C 180,E1 -28010.141,E2 -28010.141} C_VEL
LIN {X 0,Y 87.972,Z 685.046,A -85,B 0,C 180,E1 -28018.643,E2 -28018.643} C_VEL
LIN {X 0,Y 95.697,Z 677.635,A -85,B 0,C 180,E1 -28025.982,E2 -28025.982} C_VEL
LIN {X 0,Y 103.324,Z 669.722,A -85,B 0,C 180,E1 -28031.544,E2 -28031.544} C_VEL
LIN {X 0,Y 111.692,Z 660.234,A -85,B 0,C 180,E1 -28036.354,E2 -28036.354} C_VEL
LIN {X 0,Y 119.293,Z 650.551,A -85,B 0,C 180,E1 -28039.985,E2 -28039.985} C_VEL
LIN {X 0,Y 127.08,Z 639.114,A -85,B 0,C 180,E1 -28043.312,E2 -28043.312} C_VEL
LIN {X 0,Y 133.805,Z 627.742,A -85,B 0,C 180,E1 -28045.817,E2 -28045.817} C_VEL
LIN {X 0,Y 140.066,Z 615.478,A -85,B 0,C 180,E1 -28047.857,E2 -28047.857} C_VEL
LIN {X 0,Y 145.678,Z 602.188,A -85,B 0,C 180,E1 -28049.581,E2 -28049.581} C_VEL
LIN {X 0,Y 150.584,Z 587.439,A -85,B 0,C 180,E1 -28051.055,E2 -28051.055} C_VEL
LIN {X 0,Y 154.268,Z 572.725,A -85,B 0,C 180,E1 -28052.134,E2 -28052.134} C_VEL
LIN {X 0,Y 156.838,Z 557.823,A -85,B 0,C 180,E1 -28052.891,E2 -28052.891} C_VEL
LIN {X 0,Y 160.343,Z 521.715,A -85,B 0,C 180,E1 -28054.254,E2 -28054.254} C_VEL
LIN {X 0,Y 158.304,Z 516.452,A -85,B 0,C 180,E1 -28057.161,E2 -28057.161} C_VEL
LIN {X 0,Y 156.298,Z 511.577,A -85,B 0,C 180,E1 -28060.623,E2 -28060.623} C_VEL
LIN {X 0,Y 154.958,Z 508.563,A -85,B 0,C 180,E1 -28063.533,E2 -28063.533} C_VEL
LIN {X 0,Y 153.864,Z 505.928,A -85,B 0,C 180,E1 -28066.797,E2 -28066.797} C_VEL
LIN {X 0,Y 152.939,Z 502.52,A -85,B 0,C 180,E1 -28073.816,E2 -28073.816} C_VEL
LIN {X 0,Y 152.976,Z 502.137,A -85,B 0,C 180,E1 -28074.727,E2 -28074.727} C_VEL
LIN {X 0,Y 152.987,Z 502.752,A -85,B 0,C 180,E1 -28076.46,E2 -28076.46} C_VEL
LIN {X 0,Y 153.817,Z 505.515,A -85,B 0,C 180,E1 -28081.854,E2 -28081.854} C_VEL
LIN {X 0,Y 154.413,Z 507.114,A -85,B 0,C 180,E1 -28083.869,E2 -28083.869} C_VEL
LIN {X 0,Y 155.368,Z 509.414,A -85,B 0,C 180,E1 -28086.33,E2 -28086.33} C_VEL
LIN {X 0,Y 156.955,Z 516.242,A -85,B 0,C 180,E1 -28090.032,E2 -28090.032} C_VEL
LIN {X 0,Y 158.679,Z 524.714,A -85,B 0,C 180,E1 -28093.364,E2 -28093.364} C_VEL
LIN {X 0,Y 159.365,Z 528.421,A -85,B 0,C 180,E1 -28094.568,E2 -28094.568} C_VEL
LIN {X 0,Y 158.873,Z 538.881,A -85,B 0,C 180,E1 -28095.428,E2 -28095.428} C_VEL
LIN {X 0,Y 154.843,Z 575.586,A -85,B 0,C 180,E1 -28096.419,E2 -28096.419} C_VEL
LIN {X 0,Y 151.833,Z 591.12,A -85,B 0,C 180,E1 -28097.035,E2 -28097.035} C_VEL
LIN {X 0,Y 147.691,Z 605.994,A -85,B 0,C 180,E1 -28097.879,E2 -28097.879} C_VEL
LIN {X 0,Y 142.178,Z 620.933,A -85,B 0,C 180,E1 -28099.028,E2 -28099.028} C_VEL
LIN {X 0,Y 136.728,Z 632.892,A -85,B 0,C 180,E1 -28100.27,E2 -28100.27} C_VEL
LIN {X 0,Y 129.001,Z 646.951,A -85,B 0,C 180,E1 -28102.156,E2 -28102.156} C_VEL
LIN {X 0,Y 120.67,Z 659.647,A -85,B 0,C 180,E1 -28104.492,E2 -28104.492} C_VEL
LIN {X 0,Y 112.768,Z 670.38,A -85,B 0,C 180,E1 -28107.365,E2 -28107.365} C_VEL
LIN {X 0,Y 104.591,Z 680.368,A -85,B 0,C 180,E1 -28111.047,E2 -28111.047} C_VEL
LIN {X 0,Y 95.666,Z 690.175,A -85,B 0,C 180,E1 -28116.089,E2 -28116.089} C_VEL
LIN {X 0,Y 87.739,Z 698.387,A -85,B 0,C 180,E1 -28122.188,E2 -28122.188} C_VEL
LIN {X 0,Y 81.092,Z 705.25,A -85,B 0,C 180,E1 -28129.457,E2 -28129.457} C_VEL
LIN {X 0,Y 75.46,Z 711.608,A -85,B 0,C 180,E1 -28139.185,E2 -28139.185} C_VEL
LIN {X 0,Y 72.251,Z 716.547,A -85,B 0,C 180,E1 -28150.094,E2 -28150.094} C_VEL
LIN {X 0,Y 71.637,Z 719.377,A -85,B 0,C 180,E1 -28158.823,E2 -28158.823} C_VEL
LIN {X 0,Y 72.8,Z 721.942,A -85,B 0,C 180,E1 -28169.998,E2 -28169.998} C_VEL
LIN {X 0,Y 72.072,Z 722.448,A -85,B 0,C 180,E1 -28175.594,E2 -28175.594} C_VEL
LIN {X 0,Y 71.866,Z 722.486,A -85,B 0,C 180,E1 -28187.058,E2 -28187.058} C_VEL
LIN {X 0,Y 74.406,Z 721.372,A -85,B 0,C 180,E1 -28198.179,E2 -28198.179} C_VEL
LIN {X 0,Y 79.619,Z 719.191,A -85,B 0,C 180,E1 -28208.159,E2 -28208.159} C_VEL
LIN {X 0,Y 86.914,Z 715.889,A -85,B 0,C 180,E1 -28216.694,E2 -28216.694} C_VEL
LIN {X 0,Y 95.977,Z 711.435,A -85,B 0,C 180,E1 -28223.653,E2 -28223.653} C_VEL
LIN {X 0,Y 106.27,Z 705.676,A -85,B 0,C 180,E1 -28229.282,E2 -28229.282} C_VEL
LIN {X 0,Y 117.557,Z 698.528,A -85,B 0,C 180,E1 -28233.729,E2 -28233.729} C_VEL
LIN {X 0,Y 128.009,Z 690.965,A -85,B 0,C 180,E1 -28236.864,E2 -28236.864} C_VEL
LIN {X 0,Y 137.202,Z 683.372,A -85,B 0,C 180,E1 -28239.194,E2 -28239.194} C_VEL
LIN {X 0,Y 148.277,Z 672.966,A -85,B 0,C 180,E1 -28241.426,E2 -28241.426} C_VEL
LIN {X 0,Y 158.006,Z 662.434,A -85,B 0,C 180,E1 -28242.992,E2 -28242.992} C_VEL
LIN {X 0,Y 167.886,Z 649.889,A -85,B 0,C 180,E1 -28244.318,E2 -28244.318} C_VEL
LIN {X 0,Y 168.288,Z 649.327,A -85,B 0,C 180,E1 -28244.358,E2 -28244.358} C_VEL
LIN {X 0,Y 171.423,Z 644.634,A -85,B 0,C 180,E1 -28244.922,E2 -28244.922} C_VEL
LIN {X 0,Y 178.829,Z 630.463,A -85,B 0,C 180,E1 -28247.537,E2 -28247.537} C_VEL
LIN {X 0,Y 181.323,Z 625.417,A -85,B 0,C 180,E1 -28248.11,E2 -28248.11} C_VEL
LIN {X 0,Y 182.197,Z 623.68,A -85,B 0,C 180,E1 -28248.209,E2 -28248.209} C_VEL
LIN {X 0,Y 188.109,Z 610.884,A -85,B 0,C 180,E1 -28248.723,E2 -28248.723} C_VEL
LIN {X 0,Y 193.195,Z 597.168,A -85,B 0,C 180,E1 -28249.161,E2 -28249.161} C_VEL
LIN {X 0,Y 197.434,Z 581.911,A -85,B 0,C 180,E1 -28249.551,E2 -28249.551} C_VEL
LIN {X 0,Y 200.287,Z 566.567,A -85,B 0,C 180,E1 -28249.867,E2 -28249.867} C_VEL
LIN {X 0,Y 200.399,Z 565.524,A -85,B 0,C 180,E1 -28249.965,E2 -28249.965} C_VEL
LIN {X 0,Y 200.188,Z 561.221,A -85,B 0,C 180,E1 -28252.438,E2 -28252.438} C_VEL
LIN {X 0,Y 200.116,Z 558.057,A -85,B 0,C 180,E1 -28255.216,E2 -28255.216} C_VEL
LIN {X 0,Y 200.164,Z 557.96,A -85,B 0,C 180,E1 -28258.24,E2 -28258.24} C_VEL
LIN {X 0,Y 200.715,Z 561.105,A -85,B 0,C 180,E1 -28262.559,E2 -28262.559} C_VEL
LIN {X 0,Y 200.878,Z 561.898,A -85,B 0,C 180,E1 -28263.279,E2 -28263.279} C_VEL
LIN {X 0,Y 198.109,Z 576.38,A -85,B 0,C 180,E1 -28263.885,E2 -28263.885} C_VEL
LIN {X 0,Y 194.294,Z 590.04,A -85,B 0,C 180,E1 -28264.541,E2 -28264.541} C_VEL
LIN {X 0,Y 189.266,Z 603.691,A -85,B 0,C 180,E1 -28265.384,E2 -28265.384} C_VEL
LIN {X 0,Y 182.909,Z 617.349,A -85,B 0,C 180,E1 -28266.505,E2 -28266.505} C_VEL
LIN {X 0,Y 175.528,Z 630.166,A -85,B 0,C 180,E1 -28267.724,E2 -28267.724} C_VEL
LIN {X 0,Y 167.297,Z 642.06,A -85,B 0,C 180,E1 -28269.188,E2 -28269.188} C_VEL
LIN {X 0,Y 158.773,Z 652.514,A -85,B 0,C 180,E1 -28270.84,E2 -28270.84} C_VEL
LIN {X 0,Y 149.545,Z 662.188,A -85,B 0,C 180,E1 -28272.808,E2 -28272.808} C_VEL
LIN {X 0,Y 138.557,Z 671.975,A -85,B 0,C 180,E1 -28275.487,E2 -28275.487} C_VEL
LIN {X 0,Y 127.865,Z 680.014,A -85,B 0,C 180,E1 -28278.543,E2 -28278.543} C_VEL
LIN {X 0,Y 117.518,Z 686.606,A -85,B 0,C 180,E1 -28282.042,E2 -28282.042} C_VEL
LIN {X 0,Y 106.314,Z 692.628,A -85,B 0,C 180,E1 -28286.825,E2 -28286.825} C_VEL
LIN {X 0,Y 98.402,Z 696.202,A -85,B 0,C 180,E1 -28291.018,E2 -28291.018} C_VEL
LIN {X 0,Y 88.771,Z 699.792,A -85,B 0,C 180,E1 -28297.661,E2 -28297.661} C_VEL
LIN {X 0,Y 80.415,Z 702.124,A -85,B 0,C 180,E1 -28305.644,E2 -28305.644} C_VEL
LIN {X 0,Y 73.749,Z 703.271,A -85,B 0,C 180,E1 -28315.129,E2 -28315.129} C_VEL
LIN {X 0,Y 69.218,Z 703.289,A -85,B 0,C 180,E1 -28326.041,E2 -28326.041} C_VEL
LIN {X 0,Y 67.008,Z 702.221,A -85,B 0,C 180,E1 -28337.894,E2 -28337.894} C_VEL
LIN {X 0,Y 67.369,Z 700.05,A -85,B 0,C 180,E1 -28350.002,E2 -28350.002} C_VEL
LIN {X 0,Y 70.25,Z 696.72,A -85,B 0,C 180,E1 -28361.544,E2 -28361.544} C_VEL
LIN {X 0,Y 75.09,Z 692.187,A -85,B 0,C 180,E1 -28371.987,E2 -28371.987} C_VEL
LIN {X 0,Y 81.895,Z 686.317,A -85,B 0,C 180,E1 -28380.992,E2 -28380.992} C_VEL
LIN {X 0,Y 90.128,Z 678.971,A -85,B 0,C 180,E1 -28388.597,E2 -28388.597} C_VEL
LIN {X 0,Y 99.424,Z 669.923,A -85,B 0,C 180,E1 -28394.982,E2 -28394.982} C_VEL
LIN {X 0,Y 108.296,Z 660.271,A -85,B 0,C 180,E1 -28399.688,E2 -28399.688} C_VEL
LIN {X 0,Y 117.637,Z 648.613,A -85,B 0,C 180,E1 -28403.758,E2 -28403.758} C_VEL
LIN {X 0,Y 125.813,Z 636.582,A -85,B 0,C 180,E1 -28406.92,E2 -28406.92} C_VEL
LIN {X 0,Y 132.909,Z 624.511,A -85,B 0,C 180,E1 -28409.235,E2 -28409.235} C_VEL
LIN {X 0,Y 139.41,Z 611.318,A -85,B 0,C 180,E1 -28411.153,E2 -28411.153} C_VEL
LIN {X 0,Y 145.213,Z 596.658,A -85,B 0,C 180,E1 -28412.786,E2 -28412.786} C_VEL
LIN {X 0,Y 149.699,Z 581.804,A -85,B 0,C 180,E1 -28414.072,E2 -28414.072} C_VEL
LIN {X 0,Y 153.038,Z 566.728,A -85,B 0,C 180,E1 -28414.963,E2 -28414.963} C_VEL
LIN {X 0,Y 155.144,Z 551.286,A -85,B 0,C 180,E1 -28415.629,E2 -28415.629} C_VEL
LIN {X 0,Y 157.676,Z 525.595,A -85,B 0,C 180,E1 -28416.523,E2 -28416.523} C_VEL
LIN {X 0,Y 155.543,Z 519.816,A -85,B 0,C 180,E1 -28420.191,E2 -28420.191} C_VEL
LIN {X 0,Y 153.885,Z 515.528,A -85,B 0,C 180,E1 -28423.925,E2 -28423.925} C_VEL
LIN {X 0,Y 152.795,Z 512.758,A -85,B 0,C 180,E1 -28427.44,E2 -28427.44} C_VEL
LIN {X 0,Y 152.078,Z 509.414,A -85,B 0,C 180,E1 -28434.363,E2 -28434.363} C_VEL
LIN {X 0,Y 152.104,Z 509.359,A -85,B 0,C 180,E1 -28435.444,E2 -28435.444} C_VEL
LIN {X 0,Y 152.681,Z 512.278,A -85,B 0,C 180,E1 -28440.933,E2 -28440.933} C_VEL
LIN {X 0,Y 153.069,Z 513.219,A -85,B 0,C 180,E1 -28442.439,E2 -28442.439} C_VEL
LIN {X 0,Y 154.005,Z 515.904,A -85,B 0,C 180,E1 -28445.318,E2 -28445.318} C_VEL
LIN {X 0,Y 155.24,Z 522.177,A -85,B 0,C 180,E1 -28448.706,E2 -28448.706} C_VEL
LIN {X 0,Y 156.565,Z 529.856,A -85,B 0,C 180,E1 -28451.735,E2 -28451.735} C_VEL
LIN {X 0,Y 156.864,Z 531.756,A -85,B 0,C 180,E1 -28452.369,E2 -28452.369} C_VEL
LIN {X 0,Y 156.495,Z 538.765,A -85,B 0,C 180,E1 -28452.975,E2 -28452.975} C_VEL
LIN {X 0,Y 152.326,Z 575.336,A -85,B 0,C 180,E1 -28453.932,E2 -28453.932} C_VEL
LIN {X 0,Y 149.278,Z 590.548,A -85,B 0,C 180,E1 -28454.517,E2 -28454.517} C_VEL
LIN {X 0,Y 144.841,Z 605.889,A -85,B 0,C 180,E1 -28455.341,E2 -28455.341} C_VEL
LIN {X 0,Y 139.203,Z 620.628,A -85,B 0,C 180,E1 -28456.412,E2 -28456.412} C_VEL
LIN {X 0,Y 132.834,Z 634.072,A -85,B 0,C 180,E1 -28457.76,E2 -28457.76} C_VEL
LIN {X 0,Y 124.886,Z 647.716,A -85,B 0,C 180,E1 -28459.533,E2 -28459.533} C_VEL
LIN {X 0,Y 116.355,Z 660.095,A -85,B 0,C 180,E1 -28461.772,E2 -28461.772} C_VEL
LIN {X 0,Y 108.18,Z 670.639,A -85,B 0,C 180,E1 -28464.56,E2 -28464.56} C_VEL
LIN {X 0,Y 98.277,Z 681.932,A -85,B 0,C 180,E1 -28468.834,E2 -28468.834} C_VEL
LIN {X 0,Y 88.888,Z 691.463,A -85,B 0,C 180,E1 -28474.124,E2 -28474.124} C_VEL
LIN {X 0,Y 79.749,Z 700.181,A -85,B 0,C 180,E1 -28481.489,E2 -28481.489} C_VEL
LIN {X 0,Y 72.404,Z 707.206,A -85,B 0,C 180,E1 -28490.53,E2 -28490.53} C_VEL
LIN {X 0,Y 67.05,Z 713.037,A -85,B 0,C 180,E1 -28501.855,E2 -28501.855} C_VEL
LIN {X 0,Y 65.003,Z 716.357,A -85,B 0,C 180,E1 -28511.071,E2 -28511.071} C_VEL
LIN {X 0,Y 64.856,Z 719.69,A -85,B 0,C 180,E1 -28523.777,E2 -28523.777} C_VEL
LIN {X 0,Y 65.661,Z 720.852,A -85,B 0,C 180,E1 -28529.998,E2 -28529.998} C_VEL
LIN {X 0,Y 64.968,Z 721.382,A -85,B 0,C 180,E1 -28536.208,E2 -28536.208} C_VEL
LIN {X 0,Y 65.023,Z 721.435,A -85,B 0,C 180,E1 -28548.917,E2 -28548.917} C_VEL
LIN {X 0,Y 68.144,Z 720.368,A -85,B 0,C 180,E1 -28561.039,E2 -28561.039} C_VEL
LIN {X 0,Y 74.079,Z 718.232,A -85,B 0,C 180,E1 -28571.609,E2 -28571.609} C_VEL
LIN {X 0,Y 82.129,Z 714.98,A -85,B 0,C 180,E1 -28580.363,E2 -28580.363} C_VEL
LIN {X 0,Y 91.891,Z 710.568,A -85,B 0,C 180,E1 -28587.272,E2 -28587.272} C_VEL
LIN {X 0,Y 102.788,Z 704.851,A -85,B 0,C 180,E1 -28592.723,E2 -28592.723} C_VEL
LIN {X 0,Y 114.575,Z 697.766,A -85,B 0,C 180,E1 -28596.933,E2 -28596.933} C_VEL
LIN {X 0,Y 125.369,Z 690.269,A -85,B 0,C 180,E1 -28599.873,E2 -28599.873} C_VEL
LIN {X 0,Y 134.838,Z 682.758,A -85,B 0,C 180,E1 -28602.023,E2 -28602.023} C_VEL
LIN {X 0,Y 144.526,Z 674.032,A -85,B 0,C 180,E1 -28603.813,E2 -28603.813} C_VEL
LIN {X 0,Y 154.41,Z 663.821,A -85,B 0,C 180,E1 -28605.274,E2 -28605.274} C_VEL
LIN {X 0,Y 164.43,Z 651.771,A -85,B 0,C 180,E1 -28606.49,E2 -28606.49} C_VEL
LIN {X 0,Y 172.86,Z 639.801,A -85,B 0,C 180,E1 -28607.351,E2 -28607.351} C_VEL
LIN {X 0,Y 179.606,Z 628.493,A -85,B 0,C 180,E1 -28608.017,E2 -28608.017} C_VEL
LIN {X 0,Y 182.197,Z 623.68,A -85,B 0,C 180,E1 -28608.209,E2 -28608.209} C_VEL
LIN {X 0,Y 184.637,Z 618.462,A -85,B 0,C 180,E1 -28608.616,E2 -28608.616} C_VEL
LIN {X 0,Y 187.925,Z 609.936,A -85,B 0,C 180,E1 -28609.802,E2 -28609.802} C_VEL
LIN {X 0,Y 190.883,Z 601.227,A -85,B 0,C 180,E1 -28610.932,E2 -28610.932} C_VEL
LIN {X 0,Y 192.66,Z 595.719,A -85,B 0,C 180,E1 -28611.295,E2 -28611.295} C_VEL
LIN {X 0,Y 196.86,Z 580.696,A -85,B 0,C 180,E1 -28611.615,E2 -28611.615} C_VEL
LIN {X 0,Y 199.046,Z 569.854,A -85,B 0,C 180,E1 -28611.881,E2 -28611.881} C_VEL
LIN {X 0,Y 199.044,Z 566.996,A -85,B 0,C 180,E1 -28613.793,E2 -28613.793} C_VEL
LIN {X 0,Y 199.104,Z 565.122,A -85,B 0,C 180,E1 -28615.445,E2 -28615.445} C_VEL
LIN {X 0,Y 199.124,Z 565.108,A -85,B 0,C 180,E1 -28618.231,E2 -28618.231} C_VEL
LIN {X 0,Y 199.274,Z 567.421,A -85,B 0,C 180,E1 -28621.463,E2 -28621.463} C_VEL
LIN {X 0,Y 196.035,Z 581.956,A -85,B 0,C 180,E1 -28622.084,E2 -28622.084} C_VEL
LIN {X 0,Y 192.248,Z 594.286,A -85,B 0,C 180,E1 -28622.656,E2 -28622.656} C_VEL
LIN {X 0,Y 186.592,Z 608.436,A -85,B 0,C 180,E1 -28623.55,E2 -28623.55} C_VEL
LIN {X 0,Y 180.217,Z 621.115,A -85,B 0,C 180,E1 -28624.537,E2 -28624.537} C_VEL
LIN {X 0,Y 173.018,Z 632.947,A -85,B 0,C 180,E1 -28625.646,E2 -28625.646} C_VEL
LIN {X 0,Y 164.625,Z 644.532,A -85,B 0,C 180,E1 -28627.011,E2 -28627.011} C_VEL
LIN {X 0,Y 154.673,Z 656.076,A -85,B 0,C 180,E1 -28628.8,E2 -28628.8} C_VEL
LIN {X 0,Y 144.859,Z 665.699,A -85,B 0,C 180,E1 -28630.764,E2 -28630.764} C_VEL
LIN {X 0,Y 133.62,Z 675.035,A -85,B 0,C 180,E1 -28633.345,E2 -28633.345} C_VEL
LIN {X 0,Y 121.712,Z 683.32,A -85,B 0,C 180,E1 -28636.599,E2 -28636.599} C_VEL
LIN {X 0,Y 112.021,Z 689.038,A -85,B 0,C 180,E1 -28639.776,E2 -28639.776} C_VEL
LIN {X 0,Y 100.435,Z 694.747,A -85,B 0,C 180,E1 -28644.546,E2 -28644.546} C_VEL
LIN {X 0,Y 89.613,Z 699.047,A -85,B 0,C 180,E1 -28650.386,E2 -28650.386} C_VEL
LIN {X 0,Y 79.845,Z 702.032,A -85,B 0,C 180,E1 -28657.615,E2 -28657.615} C_VEL
LIN {X 0,Y 71.477,Z 703.81,A -85,B 0,C 180,E1 -28666.511,E2 -28666.511} C_VEL
LIN {X 0,Y 65.061,Z 704.439,A -85,B 0,C 180,E1 -28677.313,E2 -28677.313} C_VEL
LIN {X 0,Y 61.118,Z 703.95,A -85,B 0,C 180,E1 -28689.823,E2 -28689.823} C_VEL
LIN {X 0,Y 59.832,Z 702.387,A -85,B 0,C 180,E1 -28703.257,E2 -28703.257} C_VEL
LIN {X 0,Y 61.482,Z 699.693,A -85,B 0,C 180,E1 -28716.566,E2 -28716.566} C_VEL
LIN {X 0,Y 65.786,Z 695.786,A -85,B 0,C 180,E1 -28728.695,E2 -28728.695} C_VEL
LIN {X 0,Y 72.086,Z 690.668,A -85,B 0,C 180,E1 -28739.176,E2 -28739.176} C_VEL
LIN {X 0,Y 80.235,Z 684.14,A -85,B 0,C 180,E1 -28747.819,E2 -28747.819} C_VEL
LIN {X 0,Y 88.346,Z 677.141,A -85,B 0,C 180,E1 -28754.114,E2 -28754.114} C_VEL
LIN {X 0,Y 97.209,Z 668.744,A -85,B 0,C 180,E1 -28759.388,E2 -28759.388} C_VEL
LIN {X 0,Y 106.662,Z 658.649,A -85,B 0,C 180,E1 -28763.819,E2 -28763.819} C_VEL
LIN {X 0,Y 115.072,Z 648.337,A -85,B 0,C 180,E1 -28767.117,E2 -28767.117} C_VEL
LIN {X 0,Y 123.592,Z 636.049,A -85,B 0,C 180,E1 -28770.133,E2 -28770.133} C_VEL
LIN {X 0,Y 130.979,Z 623.629,A -85,B 0,C 180,E1 -28772.294,E2 -28772.294} C_VEL
LIN {X 0,Y 137.692,Z 610,A -85,B 0,C 180,E1 -28774.106,E2 -28774.106} C_VEL
LIN {X 0,Y 143.3,Z 595.782,A -85,B 0,C 180,E1 -28775.557,E2 -28775.557} C_VEL
LIN {X 0,Y 147.718,Z 581.125,A -85,B 0,C 180,E1 -28776.723,E2 -28776.723} C_VEL
LIN {X 0,Y 151.046,Z 565.898,A -85,B 0,C 180,E1 -28777.538,E2 -28777.538} C_VEL
LIN {X 0,Y 153.163,Z 549.696,A -85,B 0,C 180,E1 -28778.216,E2 -28778.216} C_VEL
LIN {X 0,Y 155.202,Z 529.54,A -85,B 0,C 180,E1 -28778.934,E2 -28778.934} C_VEL
LIN {X 0,Y 153.484,Z 524.477,A -85,B 0,C 180,E1 -28782.551,E2 -28782.551} C_VEL
LIN {X 0,Y 152.492,Z 521.749,A -85,B 0,C 180,E1 -28785.26,E2 -28785.26} C_VEL
LIN {X 0,Y 151.746,Z 519.599,A -85,B 0,C 180,E1 -28788.092,E2 -28788.092} C_VEL
LIN {X 0,Y 151.211,Z 516.446,A -85,B 0,C 180,E1 -28794.666,E2 -28794.666} C_VEL
LIN {X 0,Y 151.205,Z 516.738,A -85,B 0,C 180,E1 -28795.668,E2 -28795.668} C_VEL
LIN {X 0,Y 151.97,Z 519.949,A -85,B 0,C 180,E1 -28801.697,E2 -28801.697} C_VEL
LIN {X 0,Y 152.673,Z 522.37,A -85,B 0,C 180,E1 -28804.239,E2 -28804.239} C_VEL
LIN {X 0,Y 153.574,Z 527.852,A -85,B 0,C 180,E1 -28807.239,E2 -28807.239} C_VEL
LIN {X 0,Y 154.589,Z 535.037,A -85,B 0,C 180,E1 -28810.084,E2 -28810.084} C_VEL
LIN {X 0,Y 154.21,Z 540.656,A -85,B 0,C 180,E1 -28810.532,E2 -28810.532} C_VEL
LIN {X 0,Y 150.277,Z 574.141,A -85,B 0,C 180,E1 -28811.342,E2 -28811.342} C_VEL
LIN {X 0,Y 147.187,Z 589.339,A -85,B 0,C 180,E1 -28811.883,E2 -28811.883} C_VEL
LIN {X 0,Y 142.696,Z 604.628,A -85,B 0,C 180,E1 -28812.634,E2 -28812.634} C_VEL
LIN {X 0,Y 137.364,Z 618.533,A -85,B 0,C 180,E1 -28813.566,E2 -28813.566} C_VEL
LIN {X 0,Y 130.806,Z 632.119,A -85,B 0,C 180,E1 -28814.737,E2 -28814.737} C_VEL
LIN {X 0,Y 123.431,Z 644.784,A -85,B 0,C 180,E1 -28816.235,E2 -28816.235} C_VEL
LIN {X 0,Y 113.887,Z 658.465,A -85,B 0,C 180,E1 -28818.414,E2 -28818.414} C_VEL
LIN {X 0,Y 105.368,Z 669.049,A -85,B 0,C 180,E1 -28820.966,E2 -28820.966} C_VEL
LIN {X 0,Y 96.461,Z 678.923,A -85,B 0,C 180,E1 -28824.394,E2 -28824.394} C_VEL
LIN {X 0,Y 86.918,Z 688.299,A -85,B 0,C 180,E1 -28829.021,E2 -28829.021} C_VEL
LIN {X 0,Y 77.534,Z 696.753,A -85,B 0,C 180,E1 -28835.332,E2 -28835.332} C_VEL
LIN {X 0,Y 68.672,Z 704.387,A -85,B 0,C 180,E1 -28844.241,E2 -28844.241} C_VEL
LIN {X 0,Y 62.029,Z 710.485,A -85,B 0,C 180,E1 -28855.491,E2 -28855.491} C_VEL
LIN {X 0,Y 58.207,Z 715.179,A -85,B 0,C 180,E1 -28868.761,E2 -28868.761} C_VEL
LIN {X 0,Y 57.715,Z 718.568,A -85,B 0,C 180,E1 -28883.003,E2 -28883.003} C_VEL
LIN {X 0,Y 58.518,Z 719.761,A -85,B 0,C 180,E1 -28889.997,E2 -28889.997} C_VEL
LIN {X 0,Y 57.871,Z 720.313,A -85,B 0,C 180,E1 -28896.972,E2 -28896.972} C_VEL
LIN {X 0,Y 58.255,Z 720.382,A -85,B 0,C 180,E1 -28911.215,E2 -28911.215} C_VEL
LIN {X 0,Y 62.091,Z 719.364,A -85,B 0,C 180,E1 -28924.464,E2 -28924.464} C_VEL
LIN {X 0,Y 68.856,Z 717.275,A -85,B 0,C 180,E1 -28935.595,E2 -28935.595} C_VEL
LIN {X 0,Y 77.727,Z 714.072,A -85,B 0,C 180,E1 -28944.461,E2 -28944.461} C_VEL
LIN {X 0,Y 89.478,Z 709.105,A -85,B 0,C 180,E1 -28951.885,E2 -28951.885} C_VEL
LIN {X 0,Y 102.689,Z 702.406,A -85,B 0,C 180,E1 -28957.501,E2 -28957.501} C_VEL
LIN {X 0,Y 115.092,Z 695.023,A -85,B 0,C 180,E1 -28961.164,E2 -28961.164} C_VEL
LIN {X 0,Y 125.955,Z 687.472,A -85,B 0,C 180,E1 -28963.693,E2 -28963.693} C_VEL
LIN {X 0,Y 137.73,Z 677.975,A -85,B 0,C 180,E1 -28965.807,E2 -28965.807} C_VEL
LIN {X 0,Y 149.39,Z 666.939,A -85,B 0,C 180,E1 -28967.457,E2 -28967.457} C_VEL
LIN {X 0,Y 160.369,Z 654.643,A -85,B 0,C 180,E1 -28968.672,E2 -28968.672} C_VEL
LIN {X 0,Y 169.729,Z 642.169,A -85,B 0,C 180,E1 -28969.539,E2 -28969.539} C_VEL
LIN {X 0,Y 178.27,Z 628.45,A -85,B 0,C 180,E1 -28970.245,E2 -28970.245} C_VEL
LIN {X 0,Y 184.27,Z 616.805,A -85,B 0,C 180,E1 -28970.689,E2 -28970.689} C_VEL
LIN {X 0,Y 190.269,Z 602.566,A -85,B 0,C 180,E1 -28971.125,E2 -28971.125} C_VEL
LIN {X 0,Y 192.66,Z 595.719,A -85,B 0,C 180,E1 -28971.295,E2 -28971.295} C_VEL
LIN {X 0,Y 193.784,Z 592.012,A -85,B 0,C 180,E1 -28971.59,E2 -28971.59} C_VEL
LIN {X 0,Y 196.358,Z 580.456,A -85,B 0,C 180,E1 -28973.503,E2 -28973.503} C_VEL
LIN {X 0,Y 197.203,Z 576.665,A -85,B 0,C 180,E1 -28973.755,E2 -28973.755} C_VEL
LIN {X 0,Y 197.672,Z 574.357,A -85,B 0,C 180,E1 -28973.814,E2 -28973.814} C_VEL
LIN {X 0,Y 197.829,Z 572.038,A -85,B 0,C 180,E1 -28975.926,E2 -28975.926} C_VEL
LIN {X 0,Y 197.794,Z 572.187,A -85,B 0,C 180,E1 -28978.219,E2 -28978.219} C_VEL
LIN {X 0,Y 197.739,Z 573.232,A -85,B 0,C 180,E1 -28979.614,E2 -28979.614} C_VEL
LIN {X 0,Y 194.336,Z 586.522,A -85,B 0,C 180,E1 -28980.159,E2 -28980.159} C_VEL
LIN {X 0,Y 189.331,Z 600.968,A -85,B 0,C 180,E1 -28980.872,E2 -28980.872} C_VEL
LIN {X 0,Y 182.814,Z 615.458,A -85,B 0,C 180,E1 -28981.837,E2 -28981.837} C_VEL
LIN {X 0,Y 175.038,Z 629.211,A -85,B 0,C 180,E1 -28982.896,E2 -28982.896} C_VEL
LIN {X 0,Y 166.462,Z 641.62,A -85,B 0,C 180,E1 -28984.134,E2 -28984.134} C_VEL
LIN {X 0,Y 156.475,Z 653.651,A -85,B 0,C 180,E1 -28985.709,E2 -28985.709} C_VEL
LIN {X 0,Y 145.356,Z 664.795,A -85,B 0,C 180,E1 -28987.636,E2 -28987.636} C_VEL
LIN {X 0,Y 133.786,Z 674.471,A -85,B 0,C 180,E1 -28989.962,E2 -28989.962} C_VEL
LIN {X 0,Y 122.434,Z 682.45,A -85,B 0,C 180,E1 -28992.634,E2 -28992.634} C_VEL
LIN {X 0,Y 109.795,Z 689.818,A -85,B 0,C 180,E1 -28996.24,E2 -28996.24} C_VEL
LIN {X 0,Y 97.669,Z 695.584,A -85,B 0,C 180,E1 -29000.708,E2 -29000.708} C_VEL
LIN {X 0,Y 86.194,Z 699.928,A -85,B 0,C 180,E1 -29006.252,E2 -29006.252} C_VEL
LIN {X 0,Y 75.682,Z 702.95,A -85,B 0,C 180,E1 -29013.311,E2 -29013.311} C_VEL
LIN {X 0,Y 66.458,Z 704.781,A -85,B 0,C 180,E1 -29022.252,E2 -29022.252} C_VEL
LIN {X 0,Y 59.166,Z 705.459,A -85,B 0,C 180,E1 -29033.569,E2 -29033.569} C_VEL
LIN {X 0,Y 54.483,Z 705.016,A -85,B 0,C 180,E1 -29047.237,E2 -29047.237} C_VEL
LIN {X 0,Y 52.803,Z 703.499,A -85,B 0,C 180,E1 -29062.354,E2 -29062.354} C_VEL
LIN {X 0,Y 54.479,Z 700.83,A -85,B 0,C 180,E1 -29077.415,E2 -29077.415} C_VEL
LIN {X 0,Y 59.172,Z 696.969,A -85,B 0,C 180,E1 -29090.877,E2 -29090.877} C_VEL
LIN {X 0,Y 66.042,Z 691.905,A -85,B 0,C 180,E1 -29102.148,E2 -29102.148} C_VEL
LIN {X 0,Y 74.815,Z 685.437,A -85,B 0,C 180,E1 -29111.116,E2 -29111.116} C_VEL
LIN {X 0,Y 82.827,Z 679.045,A -85,B 0,C 180,E1 -29117.043,E2 -29117.043} C_VEL
LIN {X 0,Y 92.805,Z 670.179,A -85,B 0,C 180,E1 -29122.67,E2 -29122.67} C_VEL
LIN {X 0,Y 102.706,Z 660.163,A -85,B 0,C 180,E1 -29126.956,E2 -29126.956} C_VEL
LIN {X 0,Y 111.444,Z 649.954,A -85,B 0,C 180,E1 -29130.125,E2 -29130.125} C_VEL
LIN {X 0,Y 119.544,Z 638.924,A -85,B 0,C 180,E1 -29132.773,E2 -29132.773} C_VEL
LIN {X 0,Y 127.129,Z 626.9,A -85,B 0,C 180,E1 -29134.856,E2 -29134.856} C_VEL
LIN {X 0,Y 134.034,Z 613.783,A -85,B 0,C 180,E1 -29136.578,E2 -29136.578} C_VEL
LIN {X 0,Y 140.195,Z 599.274,A -85,B 0,C 180,E1 -29138.033,E2 -29138.033} C_VEL
LIN {X 0,Y 144.796,Z 585.167,A -85,B 0,C 180,E1 -29139.171,E2 -29139.171} C_VEL
LIN {X 0,Y 148.458,Z 570.094,A -85,B 0,C 180,E1 -29139.977,E2 -29139.977} C_VEL
LIN {X 0,Y 150.873,Z 554.249,A -85,B 0,C 180,E1 -29140.626,E2 -29140.626} C_VEL
LIN {X 0,Y 153.019,Z 533.837,A -85,B 0,C 180,E1 -29141.332,E2 -29141.332} C_VEL
LIN {X 0,Y 151.779,Z 529.809,A -85,B 0,C 180,E1 -29144.591,E2 -29144.591} C_VEL
LIN {X 0,Y 150.766,Z 526.548,A -85,B 0,C 180,E1 -29148.509,E2 -29148.509} C_VEL
LIN {X 0,Y 150.323,Z 523.648,A -85,B 0,C 180,E1 -29154.634,E2 -29154.634} C_VEL
LIN {X 0,Y 150.307,Z 524.268,A -85,B 0,C 180,E1 -29156.145,E2 -29156.145} C_VEL
LIN {X 0,Y 150.94,Z 526.875,A -85,B 0,C 180,E1 -29161.167,E2 -29161.167} C_VEL
LIN {X 0,Y 151.405,Z 528.803,A -85,B 0,C 180,E1 -29163.156,E2 -29163.156} C_VEL
LIN {X 0,Y 152.046,Z 533.865,A -85,B 0,C 180,E1 -29165.886,E2 -29165.886} C_VEL
LIN {X 0,Y 152.566,Z 538.564,A -85,B 0,C 180,E1 -29167.802,E2 -29167.802} C_VEL
LIN {X 0,Y 152.017,Z 544.114,A -85,B 0,C 180,E1 -29168.047,E2 -29168.047} C_VEL
LIN {X 0,Y 148.475,Z 573.266,A -85,B 0,C 180,E1 -29168.71,E2 -29168.71} C_VEL
LIN {X 0,Y 145.188,Z 588.915,A -85,B 0,C 180,E1 -29169.219,E2 -29169.219} C_VEL
LIN {X 0,Y 140.456,Z 604.466,A -85,B 0,C 180,E1 -29169.904,E2 -29169.904} C_VEL
LIN {X 0,Y 135.022,Z 618.206,A -85,B 0,C 180,E1 -29170.75,E2 -29170.75} C_VEL
LIN {X 0,Y 128.334,Z 631.688,A -85,B 0,C 180,E1 -29171.794,E2 -29171.794} C_VEL
LIN {X 0,Y 120.046,Z 645.4,A -85,B 0,C 180,E1 -29173.276,E2 -29173.276} C_VEL
LIN {X 0,Y 110.974,Z 657.904,A -85,B 0,C 180,E1 -29175.131,E2 -29175.131} C_VEL
LIN {X 0,Y 101.436,Z 669.284,A -85,B 0,C 180,E1 -29177.697,E2 -29177.697} C_VEL
LIN {X 0,Y 90.684,Z 680.447,A -85,B 0,C 180,E1 -29181.565,E2 -29181.565} C_VEL
LIN {X 0,Y 80.379,Z 689.764,A -85,B 0,C 180,E1 -29186.399,E2 -29186.399} C_VEL
LIN {X 0,Y 70.979,Z 697.518,A -85,B 0,C 180,E1 -29192.685,E2 -29192.685} C_VEL
LIN {X 0,Y 61.697,Z 704.816,A -85,B 0,C 180,E1 -29202.235,E2 -29202.235} C_VEL
LIN {X 0,Y 54.726,Z 710.591,A -85,B 0,C 180,E1 -29214.695,E2 -29214.695} C_VEL
LIN {X 0,Y 51.521,Z 713.998,A -85,B 0,C 180,E1 -29225.841,E2 -29225.841} C_VEL
LIN {X 0,Y 50.576,Z 717.445,A -85,B 0,C 180,E1 -29242.01,E2 -29242.01} C_VEL
LIN {X 0,Y 51.369,Z 718.67,A -85,B 0,C 180,E1 -29249.997,E2 -29249.997} C_VEL
LIN {X 0,Y 50.772,Z 719.23,A -85,B 0,C 180,E1 -29257.953,E2 -29257.953} C_VEL
LIN {X 0,Y 51.602,Z 719.329,A -85,B 0,C 180,E1 -29274.112,E2 -29274.112} C_VEL
LIN {X 0,Y 56.297,Z 718.359,A -85,B 0,C 180,E1 -29288.618,E2 -29288.618} C_VEL
LIN {X 0,Y 64.007,Z 716.315,A -85,B 0,C 180,E1 -29300.223,E2 -29300.223} C_VEL
LIN {X 0,Y 73.772,Z 713.162,A -85,B 0,C 180,E1 -29309.019,E2 -29309.019} C_VEL
LIN {X 0,Y 85.545,Z 708.58,A -85,B 0,C 180,E1 -29315.747,E2 -29315.747} C_VEL
LIN {X 0,Y 97.045,Z 703.213,A -85,B 0,C 180,E1 -29320.289,E2 -29320.289} C_VEL
LIN {X 0,Y 109.747,Z 696.253,A -85,B 0,C 180,E1 -29323.848,E2 -29323.848} C_VEL
LIN {X 0,Y 121.173,Z 688.885,A -85,B 0,C 180,E1 -29326.275,E2 -29326.275} C_VEL
LIN {X 0,Y 132.801,Z 680.141,A -85,B 0,C 180,E1 -29328.236,E2 -29328.236} C_VEL
LIN {X 0,Y 144.605,Z 669.729,A -85,B 0,C 180,E1 -29329.779,E2 -29329.779} C_VEL
LIN {X 0,Y 154.843,Z 659.187,A -85,B 0,C 180,E1 -29330.803,E2 -29330.803} C_VEL
LIN {X 0,Y 165.143,Z 646.624,A -85,B 0,C 180,E1 -29331.654,E2 -29331.654} C_VEL
LIN {X 0,Y 173.75,Z 634.089,A -85,B 0,C 180,E1 -29332.288,E2 -29332.288} C_VEL
LIN {X 0,Y 181.538,Z 620.417,A -85,B 0,C 180,E1 -29332.746,E2 -29332.746} C_VEL
LIN {X 0,Y 186.724,Z 609.313,A -85,B 0,C 180,E1 -29333.059,E2 -29333.059} C_VEL
LIN {X 0,Y 192.114,Z 595.119,A -85,B 0,C 180,E1 -29333.413,E2 -29333.413} C_VEL
LIN {X 0,Y 196.452,Z 579.847,A -85,B 0,C 180,E1 -29333.698,E2 -29333.698} C_VEL
LIN {X 0,Y 197.203,Z 576.665,A -85,B 0,C 180,E1 -29333.755,E2 -29333.755} C_VEL
LIN {X 0,Y 197.284,Z 576.116,A -85,B 0,C 180,E1 -29334.034,E2 -29334.034} C_VEL
LIN {X 0,Y 196.971,Z 576.965,A -85,B 0,C 180,E1 -29334.762,E2 -29334.762} C_VEL
LIN {X 0,Y 196.043,Z 580.241,A -85,B 0,C 180,E1 -29335.833,E2 -29335.833} C_VEL
LIN {X 0,Y 194.31,Z 586.14,A -85,B 0,C 180,E1 -29336.964,E2 -29336.964} C_VEL
LIN {X 0,Y 192.038,Z 593.3,A -85,B 0,C 180,E1 -29338.051,E2 -29338.051} C_VEL
LIN {X 0,Y 190.235,Z 598.275,A -85,B 0,C 180,E1 -29338.542,E2 -29338.542} C_VEL
LIN {X 0,Y 189.247,Z 600.817,A -85,B 0,C 180,E1 -29338.692,E2 -29338.692} C_VEL
LIN {X 0,Y 183.607,Z 613.567,A -85,B 0,C 180,E1 -29339.463,E2 -29339.463} C_VEL
LIN {X 0,Y 176.696,Z 626.264,A -85,B 0,C 180,E1 -29340.311,E2 -29340.311} C_VEL
LIN {X 0,Y 168.71,Z 638.388,A -85,B 0,C 180,E1 -29341.322,E2 -29341.322} C_VEL
LIN {X 0,Y 159.733,Z 649.79,A -85,B 0,C 180,E1 -29342.522,E2 -29342.522} C_VEL
LIN {X 0,Y 149.702,Z 660.51,A -85,B 0,C 180,E1 -29343.993,E2 -29343.993} C_VEL
LIN {X 0,Y 138.756,Z 670.357,A -85,B 0,C 180,E1 -29345.815,E2 -29345.815} C_VEL
LIN {X 0,Y 127.703,Z 678.722,A -85,B 0,C 180,E1 -29347.878,E2 -29347.878} C_VEL
LIN {X 0,Y 116.094,Z 686.125,A -85,B 0,C 180,E1 -29350.465,E2 -29350.465} C_VEL
LIN {X 0,Y 104.802,Z 692.145,A -85,B 0,C 180,E1 -29353.513,E2 -29353.513} C_VEL
LIN {X 0,Y 92.758,Z 697.416,A -85,B 0,C 180,E1 -29357.643,E2 -29357.643} C_VEL
LIN {X 0,Y 83.263,Z 700.796,A -85,B 0,C 180,E1 -29361.81,E2 -29361.81} C_VEL
LIN {X 0,Y 71.983,Z 703.872,A -85,B 0,C 180,E1 -29368.52,E2 -29368.52} C_VEL
LIN {X 0,Y 61.867,Z 705.751,A -85,B 0,C 180,E1 -29377.333,E2 -29377.333} C_VEL
LIN {X 0,Y 53.574,Z 706.479,A -85,B 0,C 180,E1 -29389.016,E2 -29389.016} C_VEL
LIN {X 0,Y 47.996,Z 706.082,A -85,B 0,C 180,E1 -29403.946,E2 -29403.946} C_VEL
LIN {X 0,Y 45.792,Z 704.605,A -85,B 0,C 180,E1 -29421.175,E2 -29421.175} C_VEL
LIN {X 0,Y 47.493,Z 701.962,A -85,B 0,C 180,E1 -29438.513,E2 -29438.513} C_VEL
LIN {X 0,Y 52.662,Z 698.151,A -85,B 0,C 180,E1 -29453.604,E2 -29453.604} C_VEL
LIN {X 0,Y 60.21,Z 693.142,A -85,B 0,C 180,E1 -29465.708,E2 -29465.708} C_VEL
LIN {X 0,Y 69.687,Z 686.732,A -85,B 0,C 180,E1 -29474.908,E2 -29474.908} C_VEL
LIN {X 0,Y 80.279,Z 678.766,A -85,B 0,C 180,E1 -29481.991,E2 -29481.991} C_VEL
LIN {X 0,Y 90.2,Z 670.284,A -85,B 0,C 180,E1 -29486.888,E2 -29486.888} C_VEL
LIN {X 0,Y 100.58,Z 660.087,A -85,B 0,C 180,E1 -29490.86,E2 -29490.86} C_VEL
LIN {X 0,Y 109.671,Z 649.668,A -85,B 0,C 180,E1 -29493.787,E2 -29493.787} C_VEL
LIN {X 0,Y 118.84,Z 637.242,A -85,B 0,C 180,E1 -29496.44,E2 -29496.44} C_VEL
LIN {X 0,Y 126.694,Z 624.648,A -85,B 0,C 180,E1 -29498.304,E2 -29498.304} C_VEL
LIN {X 0,Y 133.803,Z 610.781,A -85,B 0,C 180,E1 -29499.864,E2 -29499.864} C_VEL
LIN {X 0,Y 139.724,Z 596.228,A -85,B 0,C 180,E1 -29501.129,E2 -29501.129} C_VEL
LIN {X 0,Y 144.22,Z 581.686,A -85,B 0,C 180,E1 -29502.13,E2 -29502.13} C_VEL
LIN {X 0,Y 147.591,Z 566.495,A -85,B 0,C 180,E1 -29502.819,E2 -29502.819} C_VEL
LIN {X 0,Y 150.101,Z 547.316,A -85,B 0,C 180,E1 -29503.509,E2 -29503.509} C_VEL
LIN {X 0,Y 151.091,Z 538.312,A -85,B 0,C 180,E1 -29503.793,E2 -29503.793} C_VEL
LIN {X 0,Y 150.168,Z 534.983,A -85,B 0,C 180,E1 -29507.027,E2 -29507.027} C_VEL
LIN {X 0,Y 149.746,Z 533.41,A -85,B 0,C 180,E1 -29509.179,E2 -29509.179} C_VEL
LIN {X 0,Y 149.433,Z 530.862,A -85,B 0,C 180,E1 -29514.602,E2 -29514.602} C_VEL
LIN {X 0,Y 149.422,Z 531.428,A -85,B 0,C 180,E1 -29516.122,E2 -29516.122} C_VEL
LIN {X 0,Y 149.901,Z 533.695,A -85,B 0,C 180,E1 -29520.503,E2 -29520.503} C_VEL
LIN {X 0,Y 150.194,Z 535.326,A -85,B 0,C 180,E1 -29522.094,E2 -29522.094} C_VEL
LIN {X 0,Y 150.602,Z 539.822,A -85,B 0,C 180,E1 -29524.485,E2 -29524.485} C_VEL
LIN {X 0,Y 150.764,Z 541.849,A -85,B 0,C 180,E1 -29525.349,E2 -29525.349} C_VEL
LIN {X 0,Y 147.046,Z 572.073,A -85,B 0,C 180,E1 -29526.001,E2 -29526.001} C_VEL
LIN {X 0,Y 143.698,Z 587.821,A -85,B 0,C 180,E1 -29526.467,E2 -29526.467} C_VEL
LIN {X 0,Y 138.972,Z 603.149,A -85,B 0,C 180,E1 -29527.043,E2 -29527.043} C_VEL
LIN {X 0,Y 133.018,Z 617.856,A -85,B 0,C 180,E1 -29527.843,E2 -29527.843} C_VEL
LIN {X 0,Y 126.213,Z 631.214,A -85,B 0,C 180,E1 -29528.743,E2 -29528.743} C_VEL
LIN {X 0,Y 117.767,Z 644.827,A -85,B 0,C 180,E1 -29530.045,E2 -29530.045} C_VEL
LIN {X 0,Y 109.138,Z 656.47,A -85,B 0,C 180,E1 -29531.533,E2 -29531.533} C_VEL
LIN {X 0,Y 99.482,Z 667.707,A -85,B 0,C 180,E1 -29533.74,E2 -29533.74} C_VEL
LIN {X 0,Y 88.279,Z 678.979,A -85,B 0,C 180,E1 -29537.188,E2 -29537.188} C_VEL
LIN {X 0,Y 78.082,Z 687.84,A -85,B 0,C 180,E1 -29541.308,E2 -29541.308} C_VEL
LIN {X 0,Y 67.357,Z 696.17,A -85,B 0,C 180,E1 -29547.513,E2 -29547.513} C_VEL
LIN {X 0,Y 57.075,Z 703.524,A -85,B 0,C 180,E1 -29556.83,E2 -29556.83} C_VEL
LIN {X 0,Y 49.003,Z 709.36,A -85,B 0,C 180,E1 -29569.802,E2 -29569.802} C_VEL
LIN {X 0,Y 45.034,Z 712.822,A -85,B 0,C 180,E1 -29582.081,E2 -29582.081} C_VEL
LIN {X 0,Y 43.455,Z 716.321,A -85,B 0,C 180,E1 -29600.689,E2 -29600.689} C_VEL
LIN {X 0,Y 44.218,Z 717.573,A -85,B 0,C 180,E1 -29609.996,E2 -29609.996} C_VEL
LIN {X 0,Y 43.692,Z 718.137,A -85,B 0,C 180,E1 -29619.253,E2 -29619.253} C_VEL
LIN {X 0,Y 45.139,Z 718.279,A -85,B 0,C 180,E1 -29637.841,E2 -29637.841} C_VEL
LIN {X 0,Y 50.863,Z 717.355,A -85,B 0,C 180,E1 -29653.694,E2 -29653.694} C_VEL
LIN {X 0,Y 59.649,Z 715.361,A -85,B 0,C 180,E1 -29665.558,E2 -29665.558} C_VEL
LIN {X 0,Y 70.336,Z 712.24,A -85,B 0,C 180,E1 -29674.056,E2 -29674.056} C_VEL
LIN {X 0,Y 82.242,Z 707.938,A -85,B 0,C 180,E1 -29680.043,E2 -29680.043} C_VEL
LIN {X 0,Y 94.859,Z 702.395,A -85,B 0,C 180,E1 -29684.387,E2 -29684.387} C_VEL
LIN {X 0,Y 107.972,Z 695.498,A -85,B 0,C 180,E1 -29687.505,E2 -29687.505} C_VEL
LIN {X 0,Y 119.665,Z 688.19,A -85,B 0,C 180,E1 -29689.636,E2 -29689.636} C_VEL
LIN {X 0,Y 131.53,Z 679.526,A -85,B 0,C 180,E1 -29691.287,E2 -29691.287} C_VEL
LIN {X 0,Y 143.515,Z 669.204,A -85,B 0,C 180,E1 -29692.573,E2 -29692.573} C_VEL
LIN {X 0,Y 153.864,Z 658.757,A -85,B 0,C 180,E1 -29693.424,E2 -29693.424} C_VEL
LIN {X 0,Y 164.261,Z 646.322,A -85,B 0,C 180,E1 -29694.111,E2 -29694.111} C_VEL
LIN {X 0,Y 172.94,Z 633.914,A -85,B 0,C 180,E1 -29694.621,E2 -29694.621} C_VEL
LIN {X 0,Y 180.78,Z 620.417,A -85,B 0,C 180,E1 -29694.974,E2 -29694.974} C_VEL
LIN {X 0,Y 186.002,Z 609.523,A -85,B 0,C 180,E1 -29695.225,E2 -29695.225} C_VEL
LIN {X 0,Y 191.829,Z 594.527,A -85,B 0,C 180,E1 -29695.536,E2 -29695.536} C_VEL
LIN {X 0,Y 196.177,Z 579.54,A -85,B 0,C 180,E1 -29695.772,E2 -29695.772} C_VEL
LIN {X 0,Y 196.277,Z 578.988,A -85,B 0,C 180,E1 -29696.102,E2 -29696.102} C_VEL
LIN {X 0,Y 196.229,Z 578.933,A -85,B 0,C 180,E1 -29697.757,E2 -29697.757} C_VEL
LIN {X 0,Y 192.262,Z 592.553,A -85,B 0,C 180,E1 -29698.311,E2 -29698.311} C_VEL
LIN {X 0,Y 189.247,Z 600.817,A -85,B 0,C 180,E1 -29698.692,E2 -29698.692} C_VEL
LIN {X 0,Y 187.003,Z 606.301,A -85,B 0,C 180,E1 -29698.768,E2 -29698.768} C_VEL
LIN {X 0,Y 182.851,Z 615.23,A -85,B 0,C 180,E1 -29698.396,E2 -29698.396} C_VEL
LIN {X 0,Y 178.211,Z 623.945,A -85,B 0,C 180,E1 -29698.033,E2 -29698.033} C_VEL
LIN {X 0,Y 175.191,Z 628.972,A -85,B 0,C 180,E1 -29698.146,E2 -29698.146} C_VEL
LIN {X 0,Y 166.929,Z 641.003,A -85,B 0,C 180,E1 -29699.081,E2 -29699.081} C_VEL
LIN {X 0,Y 157.5,Z 652.485,A -85,B 0,C 180,E1 -29700.196,E2 -29700.196} C_VEL
LIN {X 0,Y 147.631,Z 662.632,A -85,B 0,C 180,E1 -29701.479,E2 -29701.479} C_VEL
LIN {X 0,Y 136.159,Z 672.553,A -85,B 0,C 180,E1 -29703.163,E2 -29703.163} C_VEL
LIN {X 0,Y 123.506,Z 681.645,A -85,B 0,C 180,E1 -29705.27,E2 -29705.27} C_VEL
LIN {X 0,Y 113.359,Z 687.795,A -85,B 0,C 180,E1 -29707.29,E2 -29707.29} C_VEL
LIN {X 0,Y 100.066,Z 694.471,A -85,B 0,C 180,E1 -29710.51,E2 -29710.51} C_VEL
LIN {X 0,Y 87.141,Z 699.615,A -85,B 0,C 180,E1 -29714.59,E2 -29714.59} C_VEL
LIN {X 0,Y 74.759,Z 703.382,A -85,B 0,C 180,E1 -29719.944,E2 -29719.944} C_VEL
LIN {X 0,Y 63.178,Z 705.9,A -85,B 0,C 180,E1 -29727.144,E2 -29727.144} C_VEL
LIN {X 0,Y 52.85,Z 707.25,A -85,B 0,C 180,E1 -29737.078,E2 -29737.078} C_VEL
LIN {X 0,Y 43.617,Z 707.371,A -85,B 0,C 180,E1 -29753.677,E2 -29753.677} C_VEL
LIN {X 0,Y 39.661,Z 706.576,A -85,B 0,C 180,E1 -29769.248,E2 -29769.248} C_VEL
LIN {X 0,Y 39.077,Z 704.54,A -85,B 0,C 180,E1 -29790.004,E2 -29790.004} C_VEL
LIN {X 0,Y 42.969,Z 701.365,A -85,B 0,C 180,E1 -29809.097,E2 -29809.097} C_VEL
LIN {X 0,Y 50.179,Z 697.022,A -85,B 0,C 180,E1 -29824.075,E2 -29824.075} C_VEL
LIN {X 0,Y 59.637,Z 691.38,A -85,B 0,C 180,E1 -29835,E2 -29835} C_VEL
LIN {X 0,Y 70.436,Z 684.286,A -85,B 0,C 180,E1 -29842.962,E2 -29842.962} C_VEL
LIN {X 0,Y 82.068,Z 675.509,A -85,B 0,C 180,E1 -29848.911,E2 -29848.911} C_VEL
LIN {X 0,Y 92.569,Z 666.309,A -85,B 0,C 180,E1 -29852.9,E2 -29852.9} C_VEL
LIN {X 0,Y 102.07,Z 656.656,A -85,B 0,C 180,E1 -29855.828,E2 -29855.828} C_VEL
LIN {X 0,Y 111.495,Z 645.423,A -85,B 0,C 180,E1 -29858.396,E2 -29858.396} C_VEL
LIN {X 0,Y 119.433,Z 634.331,A -85,B 0,C 180,E1 -29860.307,E2 -29860.307} C_VEL
LIN {X 0,Y 127.521,Z 620.863,A -85,B 0,C 180,E1 -29861.932,E2 -29861.932} C_VEL
LIN {X 0,Y 134.004,Z 607.656,A -85,B 0,C 180,E1 -29863.163,E2 -29863.163} C_VEL
LIN {X 0,Y 139.44,Z 593.725,A -85,B 0,C 180,E1 -29864.198,E2 -29864.198} C_VEL
LIN {X 0,Y 143.457,Z 580.183,A -85,B 0,C 180,E1 -29865.007,E2 -29865.007} C_VEL
LIN {X 0,Y 146.748,Z 564.615,A -85,B 0,C 180,E1 -29865.613,E2 -29865.613} C_VEL
LIN {X 0,Y 149.392,Z 543,A -85,B 0,C 180,E1 -29866.395,E2 -29866.395} C_VEL
LIN {X 0,Y 148.806,Z 540.368,A -85,B 0,C 180,E1 -29869.523,E2 -29869.523} C_VEL
LIN {X 0,Y 148.545,Z 538.062,A -85,B 0,C 180,E1 -29874.57,E2 -29874.57} C_VEL
LIN {X 0,Y 148.582,Z 539.176,A -85,B 0,C 180,E1 -29877.288,E2 -29877.288} C_VEL
LIN {X 0,Y 148.888,Z 540.508,A -85,B 0,C 180,E1 -29879.852,E2 -29879.852} C_VEL
LIN {X 0,Y 149.044,Z 541.976,A -85,B 0,C 180,E1 -29881.097,E2 -29881.097} C_VEL
LIN {X 0,Y 149.215,Z 545.101,A -85,B 0,C 180,E1 -29882.749,E2 -29882.749} C_VEL
LIN {X 0,Y 145.857,Z 571.373,A -85,B 0,C 180,E1 -29883.247,E2 -29883.247} C_VEL
LIN {X 0,Y 142.532,Z 586.761,A -85,B 0,C 180,E1 -29883.656,E2 -29883.656} C_VEL
LIN {X 0,Y 137.841,Z 601.828,A -85,B 0,C 180,E1 -29884.123,E2 -29884.123} C_VEL
LIN {X 0,Y 132.232,Z 615.714,A -85,B 0,C 180,E1 -29884.769,E2 -29884.769} C_VEL
LIN {X 0,Y 125.318,Z 629.244,A -85,B 0,C 180,E1 -29885.475,E2 -29885.475} C_VEL
LIN {X 0,Y 116.735,Z 643.067,A -85,B 0,C 180,E1 -29886.599,E2 -29886.599} C_VEL
LIN {X 0,Y 107.697,Z 655.092,A -85,B 0,C 180,E1 -29887.85,E2 -29887.85} C_VEL
LIN {X 0,Y 98.016,Z 666.104,A -85,B 0,C 180,E1 -29889.63,E2 -29889.63} C_VEL
LIN {X 0,Y 86.422,Z 677.494,A -85,B 0,C 180,E1 -29892.612,E2 -29892.612} C_VEL
LIN {X 0,Y 76.07,Z 686.162,A -85,B 0,C 180,E1 -29896.09,E2 -29896.09} C_VEL
LIN {X 0,Y 64.316,Z 694.801,A -85,B 0,C 180,E1 -29901.746,E2 -29901.746} C_VEL
LIN {X 0,Y 53.047,Z 702.225,A -85,B 0,C 180,E1 -29910.549,E2 -29910.549} C_VEL
LIN {X 0,Y 43.731,Z 708.125,A -85,B 0,C 180,E1 -29923.678,E2 -29923.678} C_VEL
LIN {X 0,Y 38.785,Z 711.64,A -85,B 0,C 180,E1 -29937.066,E2 -29937.066} C_VEL
LIN {X 0,Y 36.358,Z 715.192,A -85,B 0,C 180,E1 -29958.85,E2 -29958.85} C_VEL
LIN {X 0,Y 37.065,Z 716.463,A -85,B 0,C 180,E1 -29969.996,E2 -29969.996} C_VEL
LIN {X 0,Y 36.706,Z 717.192,A -85,B 0,C 180,E1 -29986.806,E2 -29986.806} C_VEL
LIN {X 0,Y 41.939,Z 716.922,A -85,B 0,C 180,E1 -30012.084,E2 -30012.084} C_VEL
LIN {X 0,Y 50.65,Z 715.518,A -85,B 0,C 180,E1 -30026.352,E2 -30026.352} C_VEL
LIN {X 0,Y 61.531,Z 713.007,A -85,B 0,C 180,E1 -30036.019,E2 -30036.019} C_VEL
LIN {X 0,Y 73.697,Z 709.336,A -85,B 0,C 180,E1 -30042.472,E2 -30042.472} C_VEL
LIN {X 0,Y 86.581,Z 704.486,A -85,B 0,C 180,E1 -30046.908,E2 -30046.908} C_VEL
LIN {X 0,Y 99.883,Z 698.339,A -85,B 0,C 180,E1 -30050.071,E2 -30050.071} C_VEL
LIN {X 0,Y 113.471,Z 690.763,A -85,B 0,C 180,E1 -30052.279,E2 -30052.279} C_VEL
LIN {X 0,Y 123.741,Z 684.026,A -85,B 0,C 180,E1 -30053.646,E2 -30053.646} C_VEL
LIN {X 0,Y 135.83,Z 674.749,A -85,B 0,C 180,E1 -30054.857,E2 -30054.857} C_VEL
LIN {X 0,Y 147.988,Z 663.704,A -85,B 0,C 180,E1 -30055.754,E2 -30055.754} C_VEL
LIN {X 0,Y 159.321,Z 651.389,A -85,B 0,C 180,E1 -30056.371,E2 -30056.371} C_VEL
LIN {X 0,Y 168.928,Z 638.895,A -85,B 0,C 180,E1 -30056.8,E2 -30056.8} C_VEL
LIN {X 0,Y 176.691,Z 626.813,A -85,B 0,C 180,E1 -30057.088,E2 -30057.088} C_VEL
LIN {X 0,Y 180.846,Z 619.372,A -85,B 0,C 180,E1 -30057.255,E2 -30057.255} C_VEL
LIN {X 0,Y 181.479,Z 618.111,A -85,B 0,C 180,E1 -30057.477,E2 -30057.477} C_VEL
LIN {X 0,Y 175.191,Z 628.972,A -85,B 0,C 180,E1 -30058.146,E2 -30058.146} C_VEL
LIN {X 0,Y 174.881,Z 630.065,A -85,B 0,C 180,E1 -30058.179,E2 -30058.179} C_VEL
LIN {X 0,Y 174.881,Z 674.003,A -85,B 0,C 180,E1 -30058.179,E2 -30058.179} C_VEL
LIN {X 0,Y 152.789,Z 674.003,A -85,B 0,C 180,E1 -30058.303,E2 -30058.303} C_VEL
LIN {X 0,Y 150.789,Z 672.003,A -85,B 0,C 180,E1 -30058.316,E2 -30058.316} C_VEL
LIN {X 0,Y 150.789,Z 664.661,A -85,B 0,C 180,E1 -30058.316,E2 -30058.316} C_VEL
LIN {X 0,Y 147.62,Z 663.15,A -85,B 0,C 180,E1 -30058.683,E2 -30058.683} C_VEL
LIN {X 0,Y 136.927,Z 672.403,A -85,B 0,C 180,E1 -30060.001,E2 -30060.001} C_VEL
LIN {X 0,Y 124.794,Z 681.206,A -85,B 0,C 180,E1 -30061.677,E2 -30061.677} C_VEL
LIN {X 0,Y 112.673,Z 688.506,A -85,B 0,C 180,E1 -30063.667,E2 -30063.667} C_VEL
LIN {X 0,Y 99.006,Z 695.25,A -85,B 0,C 180,E1 -30066.411,E2 -30066.411} C_VEL
LIN {X 0,Y 85.616,Z 700.451,A -85,B 0,C 180,E1 -30069.939,E2 -30069.939} C_VEL
LIN {X 0,Y 72.62,Z 704.277,A -85,B 0,C 180,E1 -30074.599,E2 -30074.599} C_VEL
LIN {X 0,Y 60.245,Z 706.844,A -85,B 0,C 180,E1 -30081.064,E2 -30081.064} C_VEL
LIN {X 0,Y 48.87,Z 708.244,A -85,B 0,C 180,E1 -30090.37,E2 -30090.37} C_VEL
LIN {X 0,Y 39.367,Z 708.502,A -85,B 0,C 180,E1 -30104.438,E2 -30104.438} C_VEL
LIN {X 0,Y 33.112,Z 707.651,A -85,B 0,C 180,E1 -30124.887,E2 -30124.887} C_VEL
LIN {X 0,Y 31.999,Z 705.65,A -85,B 0,C 180,E1 -30150.005,E2 -30150.005} C_VEL
LIN {X 0,Y 36.382,Z 702.522,A -85,B 0,C 180,E1 -30172.731,E2 -30172.731} C_VEL
LIN {X 0,Y 44.54,Z 698.229,A -85,B 0,C 180,E1 -30189.14,E2 -30189.14} C_VEL
LIN {X 0,Y 54.893,Z 692.647,A -85,B 0,C 180,E1 -30200.194,E2 -30200.194} C_VEL
LIN {X 0,Y 66.456,Z 685.612,A -85,B 0,C 180,E1 -30207.785,E2 -30207.785} C_VEL
LIN {X 0,Y 78.692,Z 676.9,A -85,B 0,C 180,E1 -30213.267,E2 -30213.267} C_VEL
LIN {X 0,Y 89.603,Z 667.782,A -85,B 0,C 180,E1 -30216.878,E2 -30216.878} C_VEL
LIN {X 0,Y 99.418,Z 658.221,A -85,B 0,C 180,E1 -30219.498,E2 -30219.498} C_VEL
LIN {X 0,Y 109.131,Z 647.093,A -85,B 0,C 180,E1 -30221.786,E2 -30221.786} C_VEL
LIN {X 0,Y 117.276,Z 636.134,A -85,B 0,C 180,E1 -30223.501,E2 -30223.501} C_VEL
LIN {X 0,Y 125.539,Z 622.859,A -85,B 0,C 180,E1 -30224.949,E2 -30224.949} C_VEL
LIN {X 0,Y 132.162,Z 609.843,A -85,B 0,C 180,E1 -30226.043,E2 -30226.043} C_VEL
LIN {X 0,Y 137.728,Z 596.145,A -85,B 0,C 180,E1 -30226.972,E2 -30226.972} C_VEL
LIN {X 0,Y 142.03,Z 582.367,A -85,B 0,C 180,E1 -30227.741,E2 -30227.741} C_VEL
LIN {X 0,Y 145.392,Z 567.381,A -85,B 0,C 180,E1 -30228.291,E2 -30228.291} C_VEL
LIN {X 0,Y 147.983,Z 548.116,A -85,B 0,C 180,E1 -30228.934,E2 -30228.934} C_VEL
LIN {X 0,Y 147.714,Z 546.853,A -85,B 0,C 180,E1 -30231.104,E2 -30231.104} C_VEL
LIN {X 0,Y 147.671,Z 545.208,A -85,B 0,C 180,E1 -30235.051,E2 -30235.051} C_VEL
LIN {X 0,Y 147.895,Z 547.437,A -85,B 0,C 180,E1 -30239.258,E2 -30239.258} C_VEL
LIN {X 0,Y 147.946,Z 548.569,A -85,B 0,C 180,E1 -30240.077,E2 -30240.077} C_VEL
LIN {X 0,Y 144.91,Z 571.205,A -85,B 0,C 180,E1 -30240.469,E2 -30240.469} C_VEL
LIN {X 0,Y 141.46,Z 586.597,A -85,B 0,C 180,E1 -30240.823,E2 -30240.823} C_VEL
LIN {X 0,Y 136.636,Z 601.663,A -85,B 0,C 180,E1 -30241.207,E2 -30241.207} C_VEL
LIN {X 0,Y 130.955,Z 615.365,A -85,B 0,C 180,E1 -30241.729,E2 -30241.729} C_VEL
LIN {X 0,Y 123.965,Z 628.791,A -85,B 0,C 180,E1 -30242.273,E2 -30242.273} C_VEL
LIN {X 0,Y 116.13,Z 641.25,A -85,B 0,C 180,E1 -30243.086,E2 -30243.086} C_VEL
LIN {X 0,Y 106.716,Z 653.691,A -85,B 0,C 180,E1 -30244.074,E2 -30244.074} C_VEL
LIN {X 0,Y 97.07,Z 664.503,A -85,B 0,C 180,E1 -30245.424,E2 -30245.424} C_VEL
LIN {X 0,Y 86.832,Z 674.452,A -85,B 0,C 180,E1 -30247.479,E2 -30247.479} C_VEL
LIN {X 0,Y 75.344,Z 684.002,A -85,B 0,C 180,E1 -30250.445,E2 -30250.445} C_VEL
LIN {X 0,Y 63.605,Z 692.388,A -85,B 0,C 180,E1 -30254.797,E2 -30254.797} C_VEL
LIN {X 0,Y 52.716,Z 699.215,A -85,B 0,C 180,E1 -30261.052,E2 -30261.052} C_VEL
LIN {X 0,Y 41.518,Z 705.537,A -85,B 0,C 180,E1 -30272.175,E2 -30272.175} C_VEL
LIN {X 0,Y 32.95,Z 710.456,A -85,B 0,C 180,E1 -30290.212,E2 -30290.212} C_VEL
LIN {X 0,Y 29.323,Z 714.049,A -85,B 0,C 180,E1 -30316.127,E2 -30316.127} C_VEL
LIN {X 0,Y 29.908,Z 715.343,A -85,B 0,C 180,E1 -30329.995,E2 -30329.995} C_VEL
LIN {X 0,Y 29.798,Z 716.099,A -85,B 0,C 180,E1 -30349.374,E2 -30349.374} C_VEL
LIN {X 0,Y 33.099,Z 716.177,A -85,B 0,C 180,E1 -30369.56,E2 -30369.56} C_VEL
LIN {X 0,Y 41.661,Z 715.352,A -85,B 0,C 180,E1 -30387.5,E2 -30387.5} C_VEL
LIN {X 0,Y 52.848,Z 713.448,A -85,B 0,C 180,E1 -30398.564,E2 -30398.564} C_VEL
LIN {X 0,Y 65.332,Z 710.386,A -85,B 0,C 180,E1 -30405.488,E2 -30405.488} C_VEL
LIN {X 0,Y 78.504,Z 706.19,A -85,B 0,C 180,E1 -30409.965,E2 -30409.965} C_VEL
LIN {X 0,Y 92.041,Z 700.763,A -85,B 0,C 180,E1 -30413.02,E2 -30413.02} C_VEL
LIN {X 0,Y 105.798,Z 693.985,A -85,B 0,C 180,E1 -30415.119,E2 -30415.119} C_VEL
LIN {X 0,Y 117.354,Z 687.193,A -85,B 0,C 180,E1 -30416.456,E2 -30416.456} C_VEL
LIN {X 0,Y 130.134,Z 678.293,A -85,B 0,C 180,E1 -30417.512,E2 -30417.512} C_VEL
LIN {X 0,Y 142.376,Z 668.139,A -85,B 0,C 180,E1 -30418.265,E2 -30418.265} C_VEL
LIN {X 0,Y 147.632,Z 663.184,A -85,B 0,C 180,E1 -30418.5,E2 -30418.5} C_VEL
LIN {X 0,Y 147.62,Z 663.15,A -85,B 0,C 180,E1 -30418.683,E2 -30418.683} C_VEL
LIN {X 0,Y 147.587,Z 665.144,A -85,B 0,C 180,E1 -30419.516,E2 -30419.516} C_VEL
LIN {X 0,Y 147.587,Z 699.151,A -85,B 0,C 180,E1 -30419.516,E2 -30419.516} C_VEL
LIN {X 0,Y 117.47,Z 699.151,A -85,B 0,C 180,E1 -30419.636,E2 -30419.636} C_VEL
LIN {X 0,Y 115.47,Z 697.151,A -85,B 0,C 180,E1 -30419.646,E2 -30419.646} C_VEL
LIN {X 0,Y 115.47,Z 690.889,A -85,B 0,C 180,E1 -30419.646,E2 -30419.646} C_VEL
LIN {X 0,Y 112.602,Z 689.131,A -85,B 0,C 180,E1 -30420.001,E2 -30420.001} C_VEL
LIN {X 0,Y 98.462,Z 696.03,A -85,B 0,C 180,E1 -30422.24,E2 -30422.24} C_VEL
LIN {X 0,Y 84.674,Z 701.287,A -85,B 0,C 180,E1 -30425.157,E2 -30425.157} C_VEL
LIN {X 0,Y 71.15,Z 705.17,A -85,B 0,C 180,E1 -30428.991,E2 -30428.991} C_VEL
LIN {X 0,Y 58.057,Z 707.788,A -85,B 0,C 180,E1 -30434.451,E2 -30434.451} C_VEL
LIN {X 0,Y 45.664,Z 709.241,A -85,B 0,C 180,E1 -30442.578,E2 -30442.578} C_VEL
LIN {X 0,Y 34.73,Z 709.549,A -85,B 0,C 180,E1 -30455.968,E2 -30455.968} C_VEL
LIN {X 0,Y 26.851,Z 708.715,A -85,B 0,C 180,E1 -30478.441,E2 -30478.441} C_VEL
LIN {X 0,Y 24.895,Z 706.764,A -85,B 0,C 180,E1 -30510.006,E2 -30510.006} C_VEL
LIN {X 0,Y 29.985,Z 703.684,A -85,B 0,C 180,E1 -30537.959,E2 -30537.959} C_VEL
LIN {X 0,Y 36.769,Z 700.643,A -85,B 0,C 180,E1 -30551.994,E2 -30551.994} C_VEL
LIN {X 0,Y 47.716,Z 695.444,A -85,B 0,C 180,E1 -30564.107,E2 -30564.107} C_VEL
LIN {X 0,Y 59.875,Z 688.837,A -85,B 0,C 180,E1 -30571.686,E2 -30571.686} C_VEL
LIN {X 0,Y 70.964,Z 681.747,A -85,B 0,C 180,E1 -30576.363,E2 -30576.363} C_VEL
LIN {X 0,Y 82.323,Z 673.254,A -85,B 0,C 180,E1 -30579.9,E2 -30579.9} C_VEL
LIN {X 0,Y 93.712,Z 663.203,A -85,B 0,C 180,E1 -30582.616,E2 -30582.616} C_VEL
LIN {X 0,Y 103.846,Z 652.61,A -85,B 0,C 180,E1 -30584.666,E2 -30584.666} C_VEL
LIN {X 0,Y 112.987,Z 641.31,A -85,B 0,C 180,E1 -30586.386,E2 -30586.386} C_VEL
LIN {X 0,Y 121.391,Z 628.956,A -85,B 0,C 180,E1 -30587.682,E2 -30587.682} C_VEL
LIN {X 0,Y 128.977,Z 615.398,A -85,B 0,C 180,E1 -30588.761,E2 -30588.761} C_VEL
LIN {X 0,Y 135.294,Z 601.287,A -85,B 0,C 180,E1 -30589.649,E2 -30589.649} C_VEL
LIN {X 0,Y 140.405,Z 586.403,A -85,B 0,C 180,E1 -30590.457,E2 -30590.457} C_VEL
LIN {X 0,Y 144.106,Z 571.476,A -85,B 0,C 180,E1 -30590.977,E2 -30590.977} C_VEL
LIN {X 0,Y 146.424,Z 556.967,A -85,B 0,C 180,E1 -30591.395,E2 -30591.395} C_VEL
LIN {X 0,Y 146.795,Z 553.782,A -85,B 0,C 180,E1 -30591.568,E2 -30591.568} C_VEL
LIN {X 0,Y 146.77,Z 552.458,A -85,B 0,C 180,E1 -30594.504,E2 -30594.504} C_VEL
LIN {X 0,Y 146.778,Z 553.154,A -85,B 0,C 180,E1 -30596.568,E2 -30596.568} C_VEL
LIN {X 0,Y 146.824,Z 553.499,A -85,B 0,C 180,E1 -30597.369,E2 -30597.369} C_VEL
LIN {X 0,Y 144.067,Z 572.319,A -85,B 0,C 180,E1 -30597.701,E2 -30597.701} C_VEL
LIN {X 0,Y 140.271,Z 588.079,A -85,B 0,C 180,E1 -30597.992,E2 -30597.992} C_VEL
LIN {X 0,Y 135.349,Z 602.653,A -85,B 0,C 180,E1 -30598.281,E2 -30598.281} C_VEL
LIN {X 0,Y 129.173,Z 616.807,A -85,B 0,C 180,E1 -30598.69,E2 -30598.69} C_VEL
LIN {X 0,Y 122.127,Z 629.769,A -85,B 0,C 180,E1 -30599.078,E2 -30599.078} C_VEL
LIN {X 0,Y 114.206,Z 641.93,A -85,B 0,C 180,E1 -30599.677,E2 -30599.677} C_VEL
LIN {X 0,Y 104.544,Z 654.269,A -85,B 0,C 180,E1 -30600.386,E2 -30600.386} C_VEL
LIN {X 0,Y 94.906,Z 664.737,A -85,B 0,C 180,E1 -30601.384,E2 -30601.384} C_VEL
LIN {X 0,Y 82.718,Z 675.992,A -85,B 0,C 180,E1 -30603.32,E2 -30603.32} C_VEL
LIN {X 0,Y 70.649,Z 685.342,A -85,B 0,C 180,E1 -30605.852,E2 -30605.852} C_VEL
LIN {X 0,Y 57.123,Z 694.143,A -85,B 0,C 180,E1 -30610.172,E2 -30610.172} C_VEL
LIN {X 0,Y 44.204,Z 701.29,A -85,B 0,C 180,E1 -30617.453,E2 -30617.453} C_VEL
LIN {X 0,Y 32.593,Z 706.956,A -85,B 0,C 180,E1 -30630.394,E2 -30630.394} C_VEL
LIN {X 0,Y 24.174,Z 711.244,A -85,B 0,C 180,E1 -30654.441,E2 -30654.441} C_VEL
LIN {X 0,Y 22.713,Z 714.217,A -85,B 0,C 180,E1 -30689.993,E2 -30689.993} C_VEL
LIN {X 0,Y 22.995,Z 714.988,A -85,B 0,C 180,E1 -30713.536,E2 -30713.536} C_VEL
LIN {X 0,Y 27.93,Z 715.126,A -85,B 0,C 180,E1 -30739.006,E2 -30739.006} C_VEL
LIN {X 0,Y 38.282,Z 714.352,A -85,B 0,C 180,E1 -30756.613,E2 -30756.613} C_VEL
LIN {X 0,Y 50.658,Z 712.475,A -85,B 0,C 180,E1 -30766.182,E2 -30766.182} C_VEL
LIN {X 0,Y 63.908,Z 709.458,A -85,B 0,C 180,E1 -30771.756,E2 -30771.756} C_VEL
LIN {X 0,Y 77.574,Z 705.315,A -85,B 0,C 180,E1 -30775.211,E2 -30775.211} C_VEL
LIN {X 0,Y 91.447,Z 699.947,A -85,B 0,C 180,E1 -30777.487,E2 -30777.487} C_VEL
LIN {X 0,Y 105.43,Z 693.229,A -85,B 0,C 180,E1 -30779.005,E2 -30779.005} C_VEL
LIN {X 0,Y 112.446,Z 689.314,A -85,B 0,C 180,E1 -30779.547,E2 -30779.547} C_VEL
